// SIMATIC STEP 7 (V5.x) project Sald_Nozzle
// CPU: CPU 315-2 DP
// station: P_ADR_BUS
// station: Hardware
// station: SIMATIC 300(1)
// program: Programma S7(1)
// program: SINAMICS_S120_CU320

FUNCTION_BLOCK FB 16
AUTHOR : Cellini
VERSION : 0.1
BEGIN
// (block stored without names or comments; labels and parameter names are numbered)
NETWORK
TITLE =
      L     DIW [AR2,P#0.0];
      SLD   3;
      T     LD 28;
      L     P#DIX 2.0;
      T     LD 36;
      L     11;
M001: T     LW 34;
      L     PIW [LD 28];
      T     DIW [LD 36];
      L     LD 28;
      L     P#2.0;
      +D;
      T     LD 28;
      L     LD 36;
      L     P#2.0;
      +D;
      T     LD 36;
      L     LW 34;
      LOOP  M001;
NETWORK
TITLE =
      A     DIX [AR2,P#10.5];
      AN    DIX [AR2,P#10.4];
      =     DIX [AR2,P#45.1];
      A     DIX [AR2,P#11.0];
      A     DIX [AR2,P#11.1];
      A     DIX [AR2,P#11.2];
      AN    DIX [AR2,P#11.3];
      A     DIX [AR2,P#11.4];
      A     DIX [AR2,P#11.5];
      A     DIX [AR2,P#10.0];
      =     DIX [AR2,P#45.2];
      A     DIX [AR2,P#17.5];
      =     DIX [AR2,P#45.3];
      A     DIX [AR2,P#23.0];
      =     DIX [AR2,P#45.4];
      A     DIX [AR2,P#23.1];
      =     DIX [AR2,P#45.5];
      A     DIX [AR2,P#23.2];
      =     DIX [AR2,P#45.6];
      A     DIX [AR2,P#15.6];
      =     DIX [AR2,P#45.7];
      A     DIX [AR2,P#15.7];
      =     DIX [AR2,P#46.0];
      L     DID [AR2,P#18.0];
      T     DID [AR2,P#62.0];
NETWORK
TITLE =
      A     DIX [AR2,P#42.0];
      =     DIX [AR2,P#33.0];
      =     DIX [AR2,P#33.1];
      =     DIX [AR2,P#33.2];
      A     M 1.1;
      =     DIX [AR2,P#33.3];
      O     DIX [AR2,P#42.2];
      O     DIX [AR2,P#11.3];
      ON    DIX [AR2,P#10.0];
      R     DIX [AR2,P#42.3];
      R     DIX [AR2,P#44.0];
      R     DIX [AR2,P#44.1];
      R     DIX [AR2,P#42.4];
      R     DIX [AR2,P#44.2];
      R     DIX [AR2,P#44.3];
      R     DIX [AR2,P#42.5];
      R     DIX [AR2,P#42.6];
      R     DIX [AR2,P#32.3];
      R     DIX [AR2,P#33.6];
      AN    DIX [AR2,P#42.2];
      =     DIX [AR2,P#33.4];
      AN    DIX [AR2,P#42.7];
      =     DIX [AR2,P#33.5];
      A     DIX [AR2,P#42.1];
      =     DIX [AR2,P#33.7];
      A     DIX [AR2,P#10.1];
      =     DIX [AR2,P#32.2];
      L     DIW [AR2,P#60.0];
      T     DIW [AR2,P#40.0];
NETWORK
TITLE =
      A     DIX [AR2,P#42.3];
      A(;
      L     DID [AR2,P#48.0];
      L     50;
      <D;
      );
      A(;
      L     DID [AR2,P#48.0];
      L     -50;
      >D;
      );
      R     DIX [AR2,P#42.3];
      A     DIX [AR2,P#42.3];
      R     DIX [AR2,P#35.0];
      S     DIX [AR2,P#35.1];
      R     DIX [AR2,P#35.2];
      R     DIX [AR2,P#35.3];
      R     DIX [AR2,P#35.4];
      R     DIX [AR2,P#35.5];
      A     DIX [AR2,P#42.3];
      AN    DIX [AR2,P#44.0];
      AN    DIX [AR2,P#44.1];
      S     DIX [AR2,P#44.0];
      JCN   M002;
      L     DID [AR2,P#48.0];
      T     DID [AR2,P#28.0];
      L     W#16#8051;
      T     DIW [AR2,P#24.0];
      L     2;
      T     DIW [AR2,P#26.0];
M002: NOP   0;
      A     DIX [AR2,P#42.3];
      A     DIX [AR2,P#44.0];
      AN    DIX [AR2,P#44.1];
      A(;
      L     DID [AR2,P#28.0];
      L     DID [AR2,P#6.0];
      ==D;
      );
      A(;
      L     W#16#5051;
      L     DIW [AR2,P#2.0];
      ==I;
      );
      A(;
      L     DIW [AR2,P#26.0];
      L     DIW [AR2,P#4.0];
      ==I;
      );
      S     DIX [AR2,P#44.1];
      A     DIX [AR2,P#42.3];
      A     DIX [AR2,P#44.0];
      A     DIX [AR2,P#44.1];
      A(;
      L     DID [AR2,P#48.0];
      L     DID [AR2,P#6.0];
      ==D;
      );
      AN    DIX [AR2,P#33.6];
      S     DIX [AR2,P#33.6];
      JCN   M003;
      L     0;
      T     DIW [AR2,P#24.0];
      T     DIW [AR2,P#26.0];
      T     DID [AR2,P#28.0];
M003: NOP   0;
      A     DIX [AR2,P#10.2];
      FP    DIX [AR2,P#47.0];
      A     DIX [AR2,P#42.3];
      A     DIX [AR2,P#44.0];
      A     DIX [AR2,P#44.1];
      A     DIX [AR2,P#33.6];
      R     DIX [AR2,P#33.6];
      R     DIX [AR2,P#42.3];
      R     DIX [AR2,P#44.0];
      R     DIX [AR2,P#44.1];
NETWORK
TITLE =
      A     DIX [AR2,P#42.4];
      AN    DIX [AR2,P#44.2];
      AN    DIX [AR2,P#44.3];
      JCN   M005;
      L     DID [AR2,P#52.0];
      L     DID [AR2,P#18.0];
      -D;
      T     DID [AR2,P#56.0];
      L     0;
      <D;
      JCN   M004;
      L     DID [AR2,P#56.0];
      NEGD;
      T     DID [AR2,P#56.0];
M004: NOP   0;
      A(;
      L     DID [AR2,P#56.0];
      L     99;
      <=D;
      );
      R     DIX [AR2,P#42.4];
M005: NOP   0;
      A     DIX [AR2,P#42.4];
      R     DIX [AR2,P#35.0];
      R     DIX [AR2,P#35.1];
      R     DIX [AR2,P#35.2];
      R     DIX [AR2,P#35.3];
      R     DIX [AR2,P#35.4];
      R     DIX [AR2,P#35.5];
      A     DIX [AR2,P#42.4];
      AN    DIX [AR2,P#44.2];
      AN    DIX [AR2,P#44.3];
      S     DIX [AR2,P#44.2];
      JCN   M006;
      L     DID [AR2,P#52.0];
      T     DID [AR2,P#28.0];
      L     W#16#8051;
      T     DIW [AR2,P#24.0];
      L     0;
      T     DIW [AR2,P#26.0];
M006: NOP   0;
      A     DIX [AR2,P#42.4];
      A     DIX [AR2,P#44.2];
      AN    DIX [AR2,P#44.3];
      A(;
      L     DID [AR2,P#28.0];
      L     DID [AR2,P#6.0];
      ==D;
      );
      A(;
      L     W#16#5051;
      L     DIW [AR2,P#2.0];
      ==I;
      );
      A(;
      L     DIW [AR2,P#26.0];
      L     DIW [AR2,P#4.0];
      ==I;
      );
      S     DIX [AR2,P#44.3];
      A     DIX [AR2,P#42.4];
      A     DIX [AR2,P#44.2];
      A     DIX [AR2,P#44.3];
      A(;
      L     DID [AR2,P#52.0];
      L     DID [AR2,P#6.0];
      ==D;
      );
      AN    DIX [AR2,P#13.0];
      AN    DIX [AR2,P#13.1];
      AN    DIX [AR2,P#13.2];
      AN    DIX [AR2,P#13.3];
      AN    DIX [AR2,P#13.4];
      AN    DIX [AR2,P#13.5];
      AN    DIX [AR2,P#33.6];
      S     DIX [AR2,P#33.6];
      JCN   M007;
      L     0;
      T     DIW [AR2,P#24.0];
      T     DIW [AR2,P#26.0];
      T     DID [AR2,P#28.0];
M007: NOP   0;
      A     DIX [AR2,P#10.2];
      FP    DIX [AR2,P#47.1];
      A     DIX [AR2,P#42.4];
      A     DIX [AR2,P#44.2];
      A     DIX [AR2,P#44.3];
      A     DIX [AR2,P#33.6];
      R     DIX [AR2,P#33.6];
      R     DIX [AR2,P#42.4];
      R     DIX [AR2,P#44.2];
      R     DIX [AR2,P#44.3];
NETWORK
TITLE =
      A     DIX [AR2,P#42.5];
      FP    DIX [AR2,P#47.2];
      A     DIX [AR2,P#45.0];
      R     DIX [AR2,P#42.5];
      A     DIX [AR2,P#42.5];
      S     DIX [AR2,P#35.0];
      R     DIX [AR2,P#35.1];
      R     DIX [AR2,P#35.2];
      R     DIX [AR2,P#35.3];
      R     DIX [AR2,P#35.4];
      R     DIX [AR2,P#35.5];
      A     DIX [AR2,P#42.5];
      A     DIX [AR2,P#13.0];
      AN    DIX [AR2,P#13.1];
      AN    DIX [AR2,P#13.2];
      AN    DIX [AR2,P#13.3];
      AN    DIX [AR2,P#13.4];
      AN    DIX [AR2,P#13.5];
      AN    DIX [AR2,P#33.6];
      S     DIX [AR2,P#33.6];
      A     DIX [AR2,P#10.2];
      FP    DIX [AR2,P#47.3];
      A     DIX [AR2,P#42.5];
      A     DIX [AR2,P#33.6];
      R     DIX [AR2,P#33.6];
      R     DIX [AR2,P#42.5];
NETWORK
TITLE =
      A     DIX [AR2,P#43.0];
      A     DIX [AR2,P#10.3];
      AN    DIX [AR2,P#15.7];
      =     DIX [AR2,P#32.1];
      A     DIX [AR2,P#43.1];
      A     DIX [AR2,P#10.3];
      AN    DIX [AR2,P#15.6];
      =     DIX [AR2,P#32.0];
NETWORK
TITLE =
      A     DIX [AR2,P#42.6];
      FP    DIX [AR2,P#47.4];
      S     DIX [AR2,P#32.3];
      A     DIX [AR2,P#10.3];
      FP    DIX [AR2,P#47.5];
      R     DIX [AR2,P#32.3];
      R     DIX [AR2,P#42.6];
NETWORK
TITLE =
      L     DIW [AR2,P#0.0];
      SLD   3;
      T     LD 28;
      L     P#DIX 24.0;
      T     LD 36;
      L     9;
M008: T     LW 34;
      L     DIW [LD 36];
      T     PQW [LD 28];
      L     LD 28;
      L     P#2.0;
      +D;
      T     LD 28;
      L     LD 36;
      L     P#2.0;
      +D;
      T     LD 36;
      L     LW 34;
      LOOP  M008;
END_FUNCTION_BLOCK

FUNCTION_BLOCK FB 20
AUTHOR : Salvati
VERSION : 0.1
BEGIN
// (block stored without names or comments; labels and parameter names are numbered)
NETWORK
TITLE =
      TAR1  LD 0;
      TAR2  LD 4;
      LAR1  P#L 8.0;
      L     B#16#10;
      T     LB [AR1,P#0.0];
      L     B#16#2;
      T     LB [AR1,P#1.0];
      L     6;
      T     LW [AR1,P#2.0];
      L     0;
      T     LW [AR1,P#4.0];
      L     DIW 0;
      SLD   3;
      L     P#I 0.0;
      +D;
      T     LD [AR1,P#6.0];
      LAR1  P#L 18.0;
      L     B#16#10;
      T     LB [AR1,P#0.0];
      L     B#16#2;
      T     LB [AR1,P#1.0];
      L     6;
      T     LW [AR1,P#2.0];
      L     0;
      T     LW [AR1,P#4.0];
      L     P#DIX 2.0;
      T     LD [AR1,P#6.0];
      BLD   7;
      UC    SFC 20;
      {     P#L 8.0, P#L 34.0, P#L 18.0 };
      BLD   8;
      LAR1  LD 0;
      LAR2  LD 4;
NETWORK
TITLE =
      TAR1  LD 0;
      TAR2  LD 4;
      LAR1  P#L 8.0;
      L     B#16#10;
      T     LB [AR1,P#0.0];
      L     B#16#2;
      T     LB [AR1,P#1.0];
      L     6;
      T     LW [AR1,P#2.0];
      L     0;
      T     LW [AR1,P#4.0];
      L     DIW 0;
      SLD   3;
      L     P#Q 0.0;
      +D;
      T     LD [AR1,P#6.0];
      LAR1  P#L 18.0;
      L     B#16#10;
      T     LB [AR1,P#0.0];
      L     B#16#2;
      T     LB [AR1,P#1.0];
      L     6;
      T     LW [AR1,P#2.0];
      L     0;
      T     LW [AR1,P#4.0];
      L     P#DIX 8.0;
      T     LD [AR1,P#6.0];
      BLD   7;
      UC    SFC 20;
      {     P#L 8.0, P#L 34.0, P#L 18.0 };
      BLD   8;
      LAR1  LD 0;
      LAR2  LD 4;
NETWORK
TITLE =
      A     DIX 14.3;
      A     M 1.5;
      JCN   M001;
      L     DIB 18;
      L     1;
      +I;
      T     DIB 18;
M001: NOP   0;
      A     DIX 14.0;
      AN    DIX 15.0;
      AN    DIX 14.3;
      S     DIX 14.3;
      R     DIX 8.4;
      JCN   M002;
      L     0;
      T     DIB 18;
M002: NOP   0;
      A     DIX 14.0;
      A     DIX 14.3;
      AN    DIX 2.4;
      AN    DIX 14.4;
      S     DIX 14.4;
      A     DIX 14.0;
      A     DIX 14.4;
      A     DIX 2.7;
      A     DIX 2.0;
      AN    DIX 14.5;
      S     DIX 14.5;
      R     DIX 14.1;
      R     DIX 14.2;
      S     DIX 8.0;
      R     DIX 8.7;
      JC    M003;
      JU    M004;
M003: NOP   0;
      L     0;
      T     DIB 10;
      T     DIB 11;
      T     DIB 13;
      L     1;
      T     DIB 12;
      L     1;
      T     DIB 9;
M004: NOP   0;
      A     DIX 14.0;
      A     DIX 14.5;
      A     DIX 2.1;
      A     DIX 2.3;
      O;
      A(;
      L     DIB 18;
      L     10;
      >=I;
      );
      R     DIX 14.3;
      R     DIX 14.4;
      R     DIX 14.5;
      R     DIX 8.0;
      R     DIX 14.0;
      S     DIX 14.2;
      JCN   M005;
      L     0;
      T     DIB 18;
M005: NOP   0;
      A     DIX 14.0;
      A     DIX 14.5;
      A     DIX 2.1;
      A     DIX 2.2;
      R     DIX 14.3;
      R     DIX 14.4;
      R     DIX 14.5;
      R     DIX 8.0;
      R     DIX 14.0;
      S     DIX 14.1;
      JC    M006;
      JU    M007;
M006: L     DIB 3;
      T     DIB 16;
M007: NOP   0;
NETWORK
TITLE =
      A     DIX 15.3;
      A     M 1.5;
      JCN   M008;
      L     DIB 18;
      L     1;
      +I;
      T     DIB 18;
M008: NOP   0;
      A     DIX 15.0;
      AN    DIX 14.0;
      AN    DIX 15.3;
      S     DIX 15.3;
      R     DIX 8.4;
      JCN   M009;
      L     0;
      T     DIB 18;
M009: NOP   0;
      A     DIX 15.0;
      A     DIX 15.3;
      AN    DIX 2.4;
      AN    DIX 15.4;
      S     DIX 15.4;
      A     DIX 15.0;
      A     DIX 15.4;
      A     DIX 2.7;
      A     DIX 2.0;
      AN    DIX 15.5;
      S     DIX 15.5;
      R     DIX 15.1;
      R     DIX 15.2;
      S     DIX 8.0;
      R     DIX 8.7;
      JC    M010;
      JU    M011;
M010: NOP   0;
      L     0;
      T     DIB 10;
      T     DIB 11;
      T     DIB 13;
      L     1;
      T     DIB 12;
      L     2;
      T     DIB 9;
M011: NOP   0;
      A     DIX 15.0;
      A     DIX 15.5;
      A     DIX 2.1;
      A     DIX 2.5;
      AN    DIX 15.6;
      S     DIX 15.6;
      S     DIX 8.6;
      JC    M012;
      JU    M013;
M012: NOP   0;
      L     DIB 17;
      T     DIB 9;
M013: NOP   0;
      A     DIX 15.0;
      A     DIX 15.6;
      A     DIX 2.1;
      A     DIX 2.3;
      O;
      A(;
      L     DIB 18;
      L     10;
      >=I;
      );
      R     DIX 15.3;
      R     DIX 15.4;
      R     DIX 15.5;
      R     DIX 15.6;
      R     DIX 8.0;
      R     DIX 8.6;
      R     DIX 15.0;
      S     DIX 15.2;
      JCN   M014;
      L     0;
      T     DIB 18;
M014: NOP   0;
      A     DIX 15.0;
      A     DIX 15.6;
      A     DIX 2.1;
      A     DIX 2.2;
      R     DIX 15.3;
      R     DIX 15.4;
      R     DIX 15.5;
      R     DIX 15.6;
      R     DIX 8.0;
      R     DIX 8.6;
      R     DIX 15.0;
      S     DIX 15.1;
NETWORK
TITLE =
      A     DIX 20.3;
      A     M 1.5;
      JCN   M015;
      L     DIB 24;
      L     1;
      +I;
      T     DIB 24;
M015: NOP   0;
      A     DIX 20.0;
      AN    DIX 21.0;
      AN    DIX 14.0;
      AN    DIX 15.0;
      AN    DIX 20.3;
      S     DIX 20.3;
      S     DIX 8.4;
      JCN   M016;
      L     0;
      T     DIB 24;
M016: NOP   0;
      A     DIX 20.0;
      A     DIX 20.3;
      A     DIX 2.4;
      AN    DIX 20.4;
      S     DIX 20.4;
      A     DIX 20.0;
      A     DIX 20.4;
      A     DIX 2.7;
      A     DIX 2.0;
      AN    DIX 20.5;
      S     DIX 20.5;
      R     DIX 20.1;
      R     DIX 20.2;
      S     DIX 8.0;
      R     DIX 8.7;
      JC    M017;
      JU    M018;
M017: NOP   0;
      L     0;
      T     DIB 10;
      T     DIB 11;
      T     DIB 13;
      L     1;
      T     DIB 12;
      L     1;
      T     DIB 9;
M018: NOP   0;
      A     DIX 20.0;
      A     DIX 20.5;
      A     DIX 2.1;
      A     DIX 2.3;
      O;
      A(;
      L     DIB 24;
      L     10;
      >=I;
      );
      R     DIX 20.3;
      R     DIX 20.4;
      R     DIX 20.5;
      R     DIX 8.0;
      R     DIX 20.0;
      S     DIX 20.2;
      JCN   M019;
      L     0;
      T     DIB 24;
M019: NOP   0;
      A     DIX 20.0;
      A     DIX 20.5;
      A     DIX 2.1;
      A     DIX 2.2;
      R     DIX 20.3;
      R     DIX 20.4;
      R     DIX 20.5;
      R     DIX 8.0;
      R     DIX 20.0;
      S     DIX 20.1;
      JC    M020;
      JU    M021;
M020: L     DIB 3;
      T     DIB 22;
M021: NOP   0;
NETWORK
TITLE =
      A     DIX 21.3;
      A     M 1.5;
      JCN   M022;
      L     DIB 24;
      L     1;
      +I;
      T     DIB 24;
M022: NOP   0;
      A     DIX 21.0;
      AN    DIX 20.0;
      AN    DIX 14.0;
      AN    DIX 15.0;
      AN    DIX 21.3;
      S     DIX 21.3;
      S     DIX 8.4;
      JCN   M023;
      L     0;
      T     DIB 24;
M023: NOP   0;
      A     DIX 21.0;
      A     DIX 21.3;
      A     DIX 2.4;
      AN    DIX 21.4;
      S     DIX 21.4;
      A     DIX 21.0;
      A     DIX 21.4;
      A     DIX 2.7;
      A     DIX 2.0;
      AN    DIX 21.5;
      S     DIX 21.5;
      R     DIX 21.1;
      R     DIX 21.2;
      S     DIX 8.0;
      R     DIX 8.7;
      JC    M024;
      JU    M025;
M024: NOP   0;
      L     0;
      T     DIB 10;
      T     DIB 11;
      T     DIB 13;
      L     1;
      T     DIB 12;
      L     2;
      T     DIB 9;
M025: NOP   0;
      A     DIX 21.0;
      A     DIX 21.5;
      A     DIX 2.1;
      A     DIX 2.5;
      AN    DIX 21.6;
      S     DIX 21.6;
      S     DIX 8.6;
      JC    M026;
      JU    M027;
M026: NOP   0;
      L     DIB 23;
      T     DIB 9;
M027: NOP   0;
      A     DIX 21.0;
      A     DIX 21.6;
      A     DIX 2.1;
      A     DIX 2.3;
      O;
      A(;
      L     DIB 24;
      L     10;
      >=I;
      );
      R     DIX 21.3;
      R     DIX 21.4;
      R     DIX 21.5;
      R     DIX 21.6;
      R     DIX 8.0;
      R     DIX 8.6;
      R     DIX 21.0;
      S     DIX 21.2;
      JCN   M028;
      L     0;
      T     DIB 24;
M028: NOP   0;
      A     DIX 21.0;
      A     DIX 21.6;
      A     DIX 2.1;
      A     DIX 2.2;
      R     DIX 21.3;
      R     DIX 21.4;
      R     DIX 21.5;
      R     DIX 21.6;
      R     DIX 8.0;
      R     DIX 8.6;
      R     DIX 21.0;
      S     DIX 21.1;
NETWORK
TITLE =
      TAR1  LD 0;
      TAR2  LD 4;
      LAR1  P#L 8.0;
      L     B#16#10;
      T     LB [AR1,P#0.0];
      L     B#16#2;
      T     LB [AR1,P#1.0];
      L     6;
      T     LW [AR1,P#2.0];
      L     0;
      T     LW [AR1,P#4.0];
      L     P#DIX 8.0;
      T     LD [AR1,P#6.0];
      LAR1  P#L 18.0;
      L     B#16#10;
      T     LB [AR1,P#0.0];
      L     B#16#2;
      T     LB [AR1,P#1.0];
      L     6;
      T     LW [AR1,P#2.0];
      L     0;
      T     LW [AR1,P#4.0];
      L     DIW 0;
      SLD   3;
      L     P#Q 0.0;
      +D;
      T     LD [AR1,P#6.0];
      BLD   7;
      UC    SFC 20;
      {     P#L 8.0, P#L 34.0, P#L 18.0 };
      BLD   8;
      LAR1  LD 0;
      LAR2  LD 4;
END_FUNCTION_BLOCK

FUNCTION_BLOCK FB 24
VERSION : 0.1
BEGIN
// (block stored without names or comments; labels and parameter names are numbered)
NETWORK
TITLE =
      L     DID [AR2,P#0.0];
      L     8;
      +I;
      SLD   3;
      T     MD 100;
      L     PIW [MD 100];
      T     DIW 52;
      L     MD 100;
      SRW   3;
      L     2;
      +D;
      SLW   3;
      T     MD 100;
      L     PIW [MD 100];
      T     DIW [AR2,P#46.0];
      L     MD 100;
      SRW   3;
      L     2;
      +D;
      SLW   3;
      T     MD 100;
      L     PIW [MD 100];
      T     DIW 64;
      L     MD 100;
      SRW   3;
      L     2;
      +D;
      SLW   3;
      T     MD 100;
      L     PIW [MD 100];
      T     DIW 62;
      L     MD 100;
      SRW   3;
      L     2;
      +D;
      SLW   3;
      T     MD 100;
      L     PID [MD 100];
      T     DID [AR2,P#36.0];
      L     MD 100;
      SRW   3;
      L     4;
      +D;
      SLW   3;
      T     MD 100;
      L     PIW [MD 100];
      T     DIW 54;
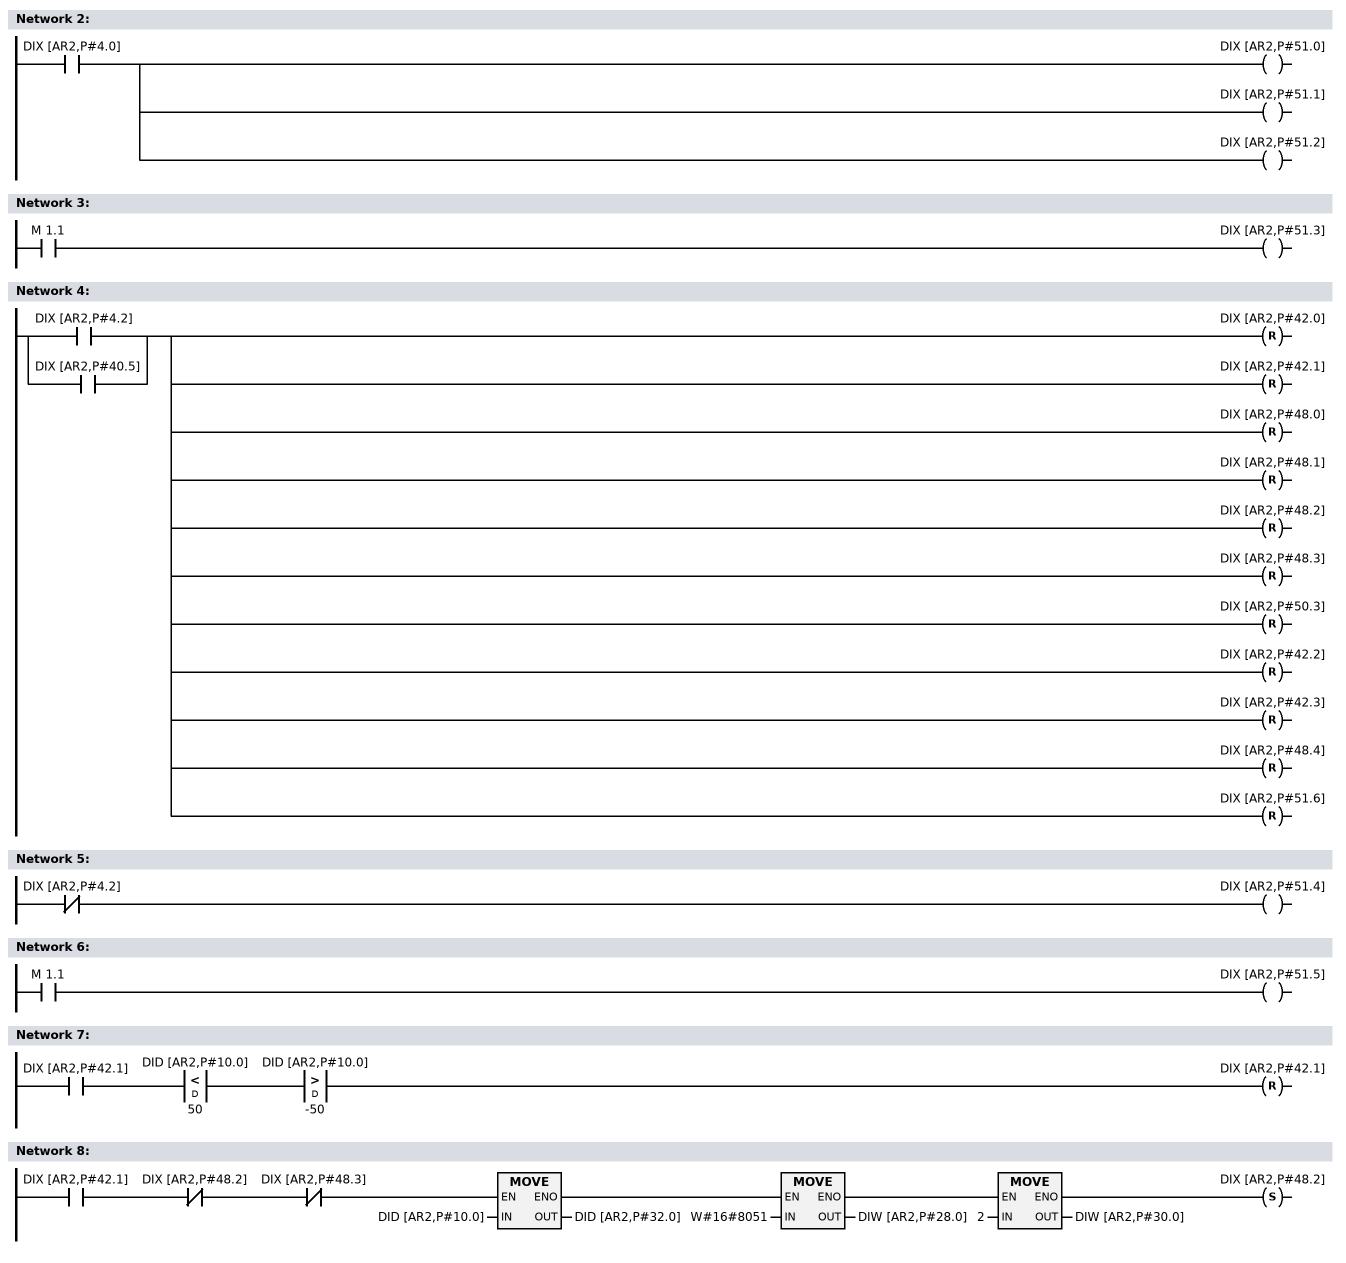
NETWORK
TITLE =
      A     DIX [AR2,P#4.0];
      =     DIX [AR2,P#51.0];
      =     DIX [AR2,P#51.1];
      =     DIX [AR2,P#51.2];
NETWORK
TITLE =
      A     M 1.1;
      =     DIX [AR2,P#51.3];
NETWORK
TITLE =
      O     DIX [AR2,P#4.2];
      O     DIX [AR2,P#40.5];
      R     DIX [AR2,P#42.0];
      R     DIX [AR2,P#42.1];
      R     DIX [AR2,P#48.0];
      R     DIX [AR2,P#48.1];
      R     DIX [AR2,P#48.2];
      R     DIX [AR2,P#48.3];
      R     DIX [AR2,P#50.3];
      R     DIX [AR2,P#42.2];
      R     DIX [AR2,P#42.3];
      R     DIX [AR2,P#48.4];
      R     DIX [AR2,P#51.6];
NETWORK
TITLE =
      AN    DIX [AR2,P#4.2];
      =     DIX [AR2,P#51.4];
NETWORK
TITLE =
      A     M 1.1;
      =     DIX [AR2,P#51.5];
NETWORK
TITLE =
      A     DIX [AR2,P#42.1];
      A(;
      L     DID [AR2,P#10.0];
      L     50;
      <D;
      );
      A(;
      L     DID [AR2,P#10.0];
      L     -50;
      >D;
      );
      R     DIX [AR2,P#42.1];
NETWORK
TITLE =
      A(;
      A(;
      A     DIX [AR2,P#42.1];
      AN    DIX [AR2,P#48.2];
      AN    DIX [AR2,P#48.3];
      JNB   M001;
      L     DID [AR2,P#10.0];
      T     DID [AR2,P#32.0];
      SET;
      SAVE;
      CLR;
M001: A     BR;
      );
      JNB   M002;
      L     W#16#8051;
      T     DIW [AR2,P#28.0];
      SET;
      SAVE;
      CLR;
M002: A     BR;
      );
      JNB   M003;
      L     2;
      T     DIW [AR2,P#30.0];
      SET;
      SAVE;
      CLR;
M003: A     BR;
      S     DIX [AR2,P#48.2];
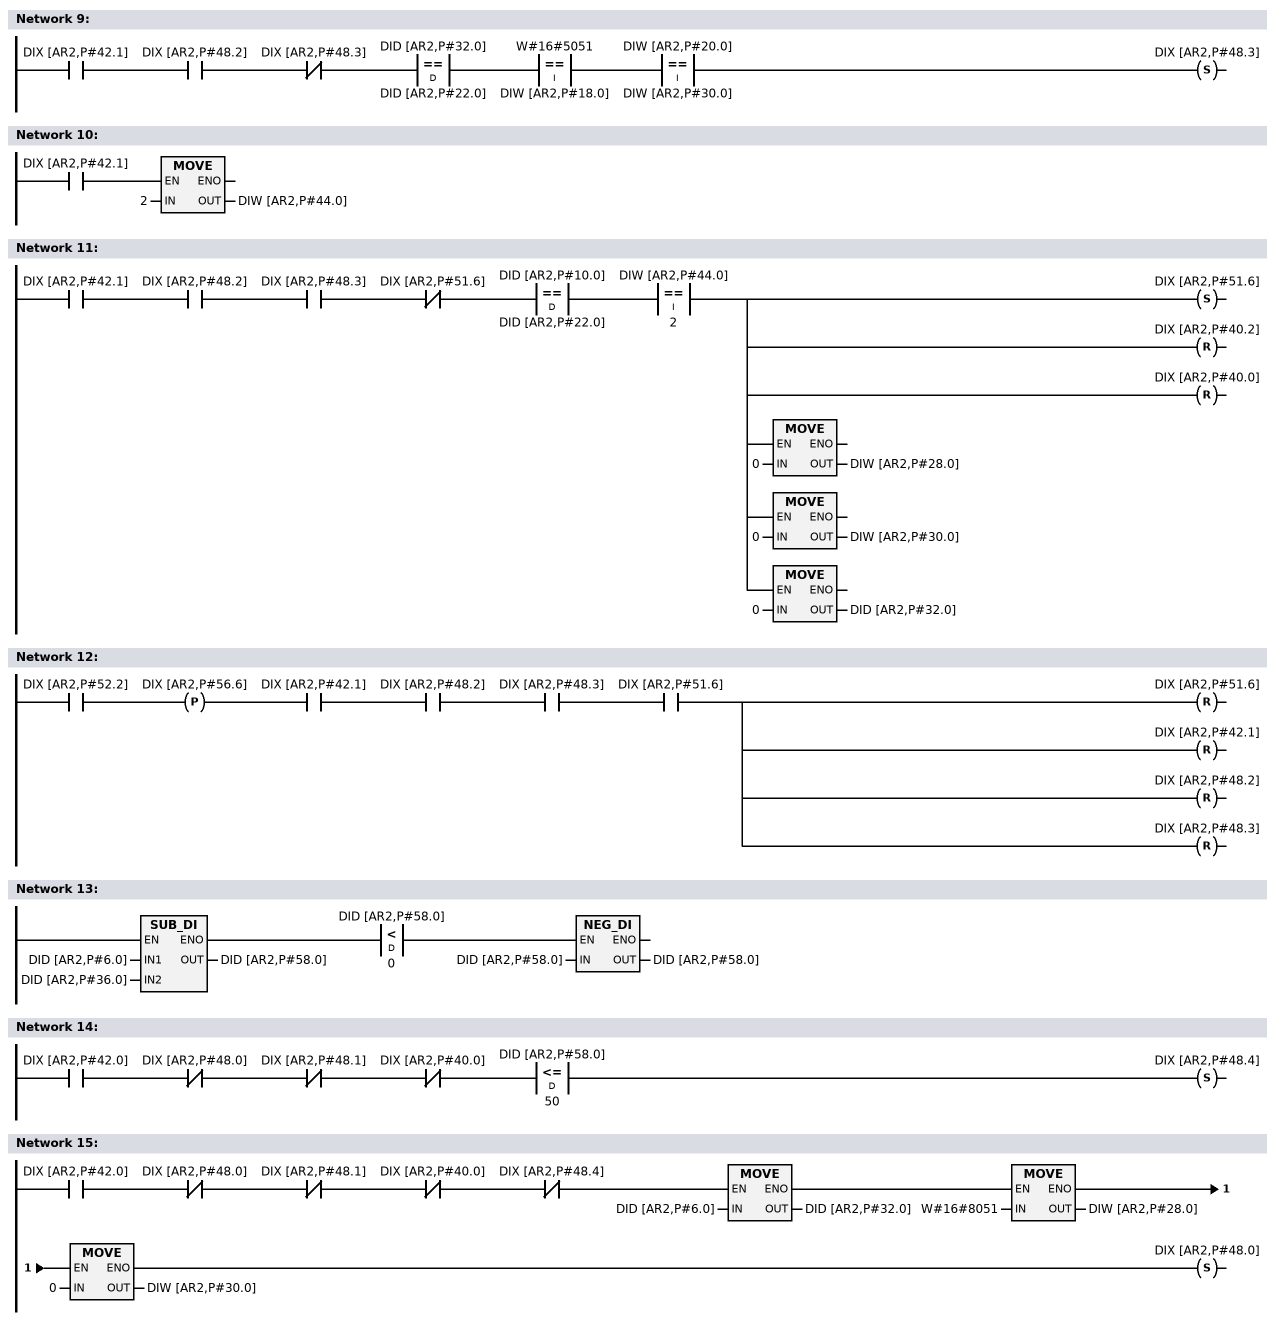
NETWORK
TITLE =
      A     DIX [AR2,P#42.1];
      A     DIX [AR2,P#48.2];
      AN    DIX [AR2,P#48.3];
      A(;
      L     DID [AR2,P#32.0];
      L     DID [AR2,P#22.0];
      ==D;
      );
      A(;
      L     W#16#5051;
      L     DIW [AR2,P#18.0];
      ==I;
      );
      A(;
      L     DIW [AR2,P#20.0];
      L     DIW [AR2,P#30.0];
      ==I;
      );
      S     DIX [AR2,P#48.3];
NETWORK
TITLE =
      A     DIX [AR2,P#42.1];
      JNB   M004;
      L     2;
      T     DIW [AR2,P#44.0];
M004: NOP   0;
NETWORK
TITLE =
      A     DIX [AR2,P#42.1];
      A     DIX [AR2,P#48.2];
      A     DIX [AR2,P#48.3];
      AN    DIX [AR2,P#51.6];
      A(;
      L     DID [AR2,P#10.0];
      L     DID [AR2,P#22.0];
      ==D;
      );
      A(;
      L     DIW [AR2,P#44.0];
      L     2;
      ==I;
      );
      =     L 0.0;
      A     L 0.0;
      BLD   102;
      S     DIX [AR2,P#51.6];
      A     L 0.0;
      BLD   102;
      R     DIX [AR2,P#40.2];
      A     L 0.0;
      BLD   102;
      R     DIX [AR2,P#40.0];
      A     L 0.0;
      JNB   M005;
      L     0;
      T     DIW [AR2,P#28.0];
M005: NOP   0;
      A     L 0.0;
      JNB   M006;
      L     0;
      T     DIW [AR2,P#30.0];
M006: NOP   0;
      A     L 0.0;
      JNB   M007;
      L     0;
      T     DID [AR2,P#32.0];
M007: NOP   0;
NETWORK
TITLE =
      A     DIX [AR2,P#52.2];
      FP    DIX [AR2,P#56.6];
      A     DIX [AR2,P#42.1];
      A     DIX [AR2,P#48.2];
      A     DIX [AR2,P#48.3];
      A     DIX [AR2,P#51.6];
      R     DIX [AR2,P#51.6];
      R     DIX [AR2,P#42.1];
      R     DIX [AR2,P#48.2];
      R     DIX [AR2,P#48.3];
NETWORK
TITLE =
      A(;
      L     DID [AR2,P#6.0];
      L     DID [AR2,P#36.0];
      -D;
      T     DID [AR2,P#58.0];
      AN    OV;
      SAVE;
      CLR;
      A     BR;
      );
      A(;
      L     DID [AR2,P#58.0];
      L     0;
      <D;
      );
      JNB   M008;
      L     DID [AR2,P#58.0];
      NEGD;
      T     DID [AR2,P#58.0];
M008: NOP   0;
NETWORK
TITLE =
      A     DIX [AR2,P#42.0];
      AN    DIX [AR2,P#48.0];
      AN    DIX [AR2,P#48.1];
      AN    DIX [AR2,P#40.0];
      A(;
      L     DID [AR2,P#58.0];
      L     50;
      <=D;
      );
      S     DIX [AR2,P#48.4];
NETWORK
TITLE =
      A(;
      A(;
      A     DIX [AR2,P#42.0];
      AN    DIX [AR2,P#48.0];
      AN    DIX [AR2,P#48.1];
      AN    DIX [AR2,P#40.0];
      AN    DIX [AR2,P#48.4];
      JNB   M009;
      L     DID [AR2,P#6.0];
      T     DID [AR2,P#32.0];
      SET;
      SAVE;
      CLR;
M009: A     BR;
      );
      JNB   M010;
      L     W#16#8051;
      T     DIW [AR2,P#28.0];
      SET;
      SAVE;
      CLR;
M010: A     BR;
      );
      JNB   M011;
      L     0;
      T     DIW [AR2,P#30.0];
      SET;
      SAVE;
      CLR;
M011: A     BR;
      S     DIX [AR2,P#48.0];
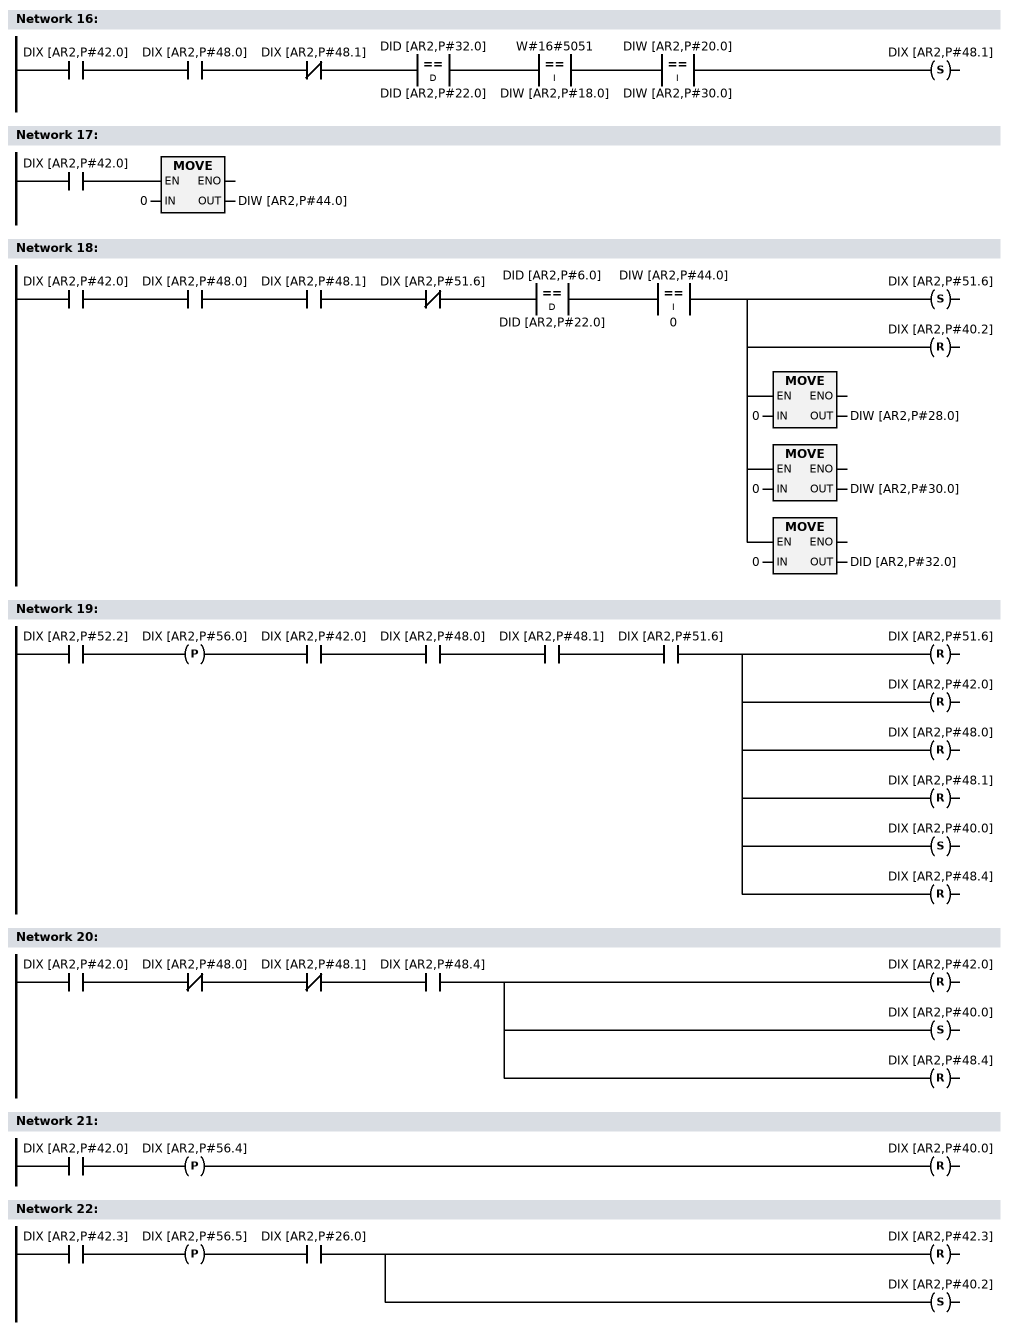
NETWORK
TITLE =
      A     DIX [AR2,P#42.0];
      A     DIX [AR2,P#48.0];
      AN    DIX [AR2,P#48.1];
      A(;
      L     DID [AR2,P#32.0];
      L     DID [AR2,P#22.0];
      ==D;
      );
      A(;
      L     W#16#5051;
      L     DIW [AR2,P#18.0];
      ==I;
      );
      A(;
      L     DIW [AR2,P#20.0];
      L     DIW [AR2,P#30.0];
      ==I;
      );
      S     DIX [AR2,P#48.1];
NETWORK
TITLE =
      A     DIX [AR2,P#42.0];
      JNB   M012;
      L     0;
      T     DIW [AR2,P#44.0];
M012: NOP   0;
NETWORK
TITLE =
      A     DIX [AR2,P#42.0];
      A     DIX [AR2,P#48.0];
      A     DIX [AR2,P#48.1];
      AN    DIX [AR2,P#51.6];
      A(;
      L     DID [AR2,P#6.0];
      L     DID [AR2,P#22.0];
      ==D;
      );
      A(;
      L     DIW [AR2,P#44.0];
      L     0;
      ==I;
      );
      =     L 0.0;
      A     L 0.0;
      BLD   102;
      S     DIX [AR2,P#51.6];
      A     L 0.0;
      BLD   102;
      R     DIX [AR2,P#40.2];
      A     L 0.0;
      JNB   M013;
      L     0;
      T     DIW [AR2,P#28.0];
M013: NOP   0;
      A     L 0.0;
      JNB   M014;
      L     0;
      T     DIW [AR2,P#30.0];
M014: NOP   0;
      A     L 0.0;
      JNB   M015;
      L     0;
      T     DID [AR2,P#32.0];
M015: NOP   0;
NETWORK
TITLE =
      A     DIX [AR2,P#52.2];
      FP    DIX [AR2,P#56.0];
      A     DIX [AR2,P#42.0];
      A     DIX [AR2,P#48.0];
      A     DIX [AR2,P#48.1];
      A     DIX [AR2,P#51.6];
      R     DIX [AR2,P#51.6];
      R     DIX [AR2,P#42.0];
      R     DIX [AR2,P#48.0];
      R     DIX [AR2,P#48.1];
      S     DIX [AR2,P#40.0];
      R     DIX [AR2,P#48.4];
NETWORK
TITLE =
      A     DIX [AR2,P#42.0];
      AN    DIX [AR2,P#48.0];
      AN    DIX [AR2,P#48.1];
      A     DIX [AR2,P#48.4];
      R     DIX [AR2,P#42.0];
      S     DIX [AR2,P#40.0];
      R     DIX [AR2,P#48.4];
NETWORK
TITLE =
      A     DIX [AR2,P#42.0];
      FP    DIX [AR2,P#56.4];
      R     DIX [AR2,P#40.0];
NETWORK
TITLE =
      A     DIX [AR2,P#42.3];
      FP    DIX [AR2,P#56.5];
      A     DIX [AR2,P#26.0];
      R     DIX [AR2,P#42.3];
      S     DIX [AR2,P#40.2];
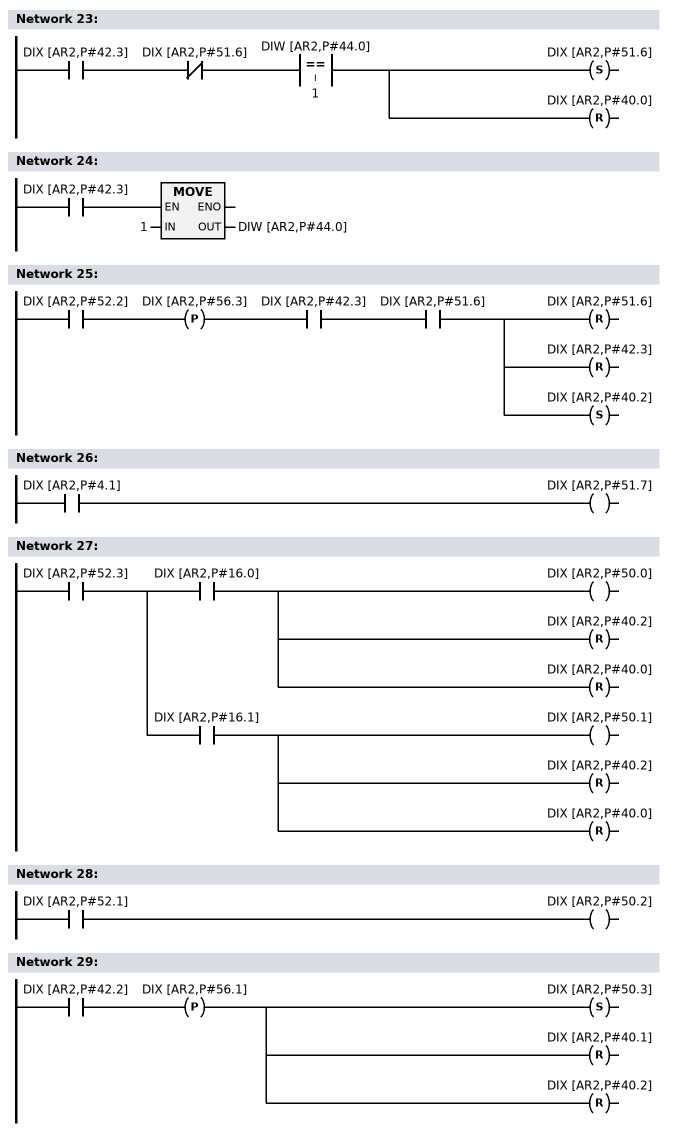
NETWORK
TITLE =
      A     DIX [AR2,P#42.3];
      AN    DIX [AR2,P#51.6];
      A(;
      L     DIW [AR2,P#44.0];
      L     1;
      ==I;
      );
      S     DIX [AR2,P#51.6];
      R     DIX [AR2,P#40.0];
NETWORK
TITLE =
      A     DIX [AR2,P#42.3];
      JNB   M016;
      L     1;
      T     DIW [AR2,P#44.0];
M016: NOP   0;
NETWORK
TITLE =
      A     DIX [AR2,P#52.2];
      FP    DIX [AR2,P#56.3];
      A     DIX [AR2,P#42.3];
      A     DIX [AR2,P#51.6];
      R     DIX [AR2,P#51.6];
      R     DIX [AR2,P#42.3];
      S     DIX [AR2,P#40.2];
NETWORK
TITLE =
      A     DIX [AR2,P#4.1];
      =     DIX [AR2,P#51.7];
NETWORK
TITLE =
      A     DIX [AR2,P#52.3];
      =     L 0.0;
      A     L 0.0;
      A     DIX [AR2,P#16.0];
      =     DIX [AR2,P#50.0];
      R     DIX [AR2,P#40.2];
      R     DIX [AR2,P#40.0];
      A     L 0.0;
      A     DIX [AR2,P#16.1];
      =     DIX [AR2,P#50.1];
      R     DIX [AR2,P#40.2];
      R     DIX [AR2,P#40.0];
NETWORK
TITLE =
      A     DIX [AR2,P#52.1];
      =     DIX [AR2,P#50.2];
NETWORK
TITLE =
      A     DIX [AR2,P#42.2];
      FP    DIX [AR2,P#56.1];
      S     DIX [AR2,P#50.3];
      R     DIX [AR2,P#40.1];
      R     DIX [AR2,P#40.2];
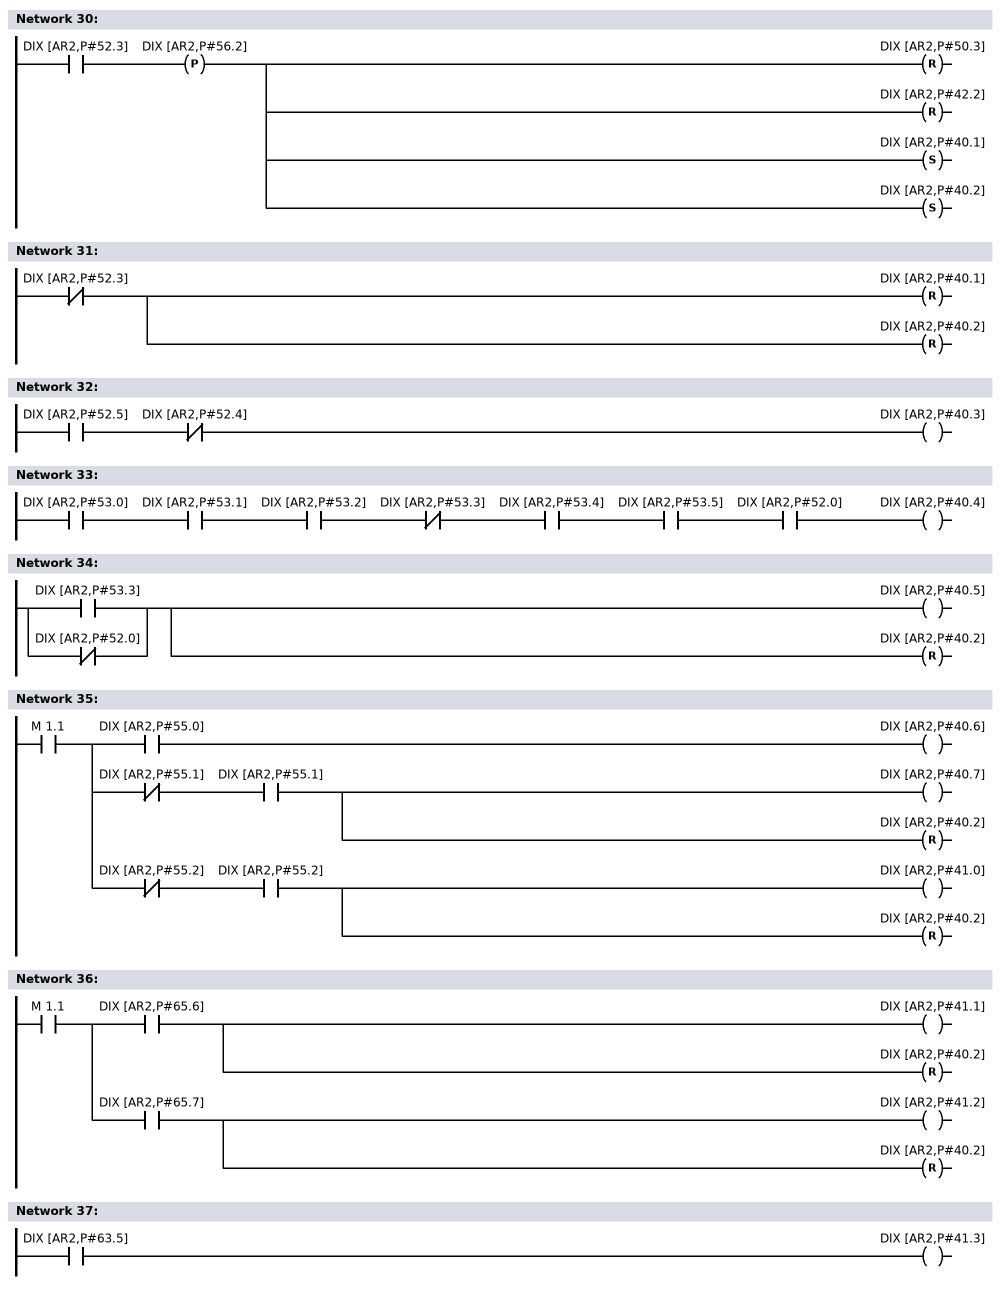
NETWORK
TITLE =
      A     DIX [AR2,P#52.3];
      FP    DIX [AR2,P#56.2];
      R     DIX [AR2,P#50.3];
      R     DIX [AR2,P#42.2];
      S     DIX [AR2,P#40.1];
      S     DIX [AR2,P#40.2];
NETWORK
TITLE =
      AN    DIX [AR2,P#52.3];
      R     DIX [AR2,P#40.1];
      R     DIX [AR2,P#40.2];
NETWORK
TITLE =
      A     DIX [AR2,P#52.5];
      AN    DIX [AR2,P#52.4];
      =     DIX [AR2,P#40.3];
NETWORK
TITLE =
      A     DIX [AR2,P#53.0];
      A     DIX [AR2,P#53.1];
      A     DIX [AR2,P#53.2];
      AN    DIX [AR2,P#53.3];
      A     DIX [AR2,P#53.4];
      A     DIX [AR2,P#53.5];
      A     DIX [AR2,P#52.0];
      =     DIX [AR2,P#40.4];
NETWORK
TITLE =
      O     DIX [AR2,P#53.3];
      ON    DIX [AR2,P#52.0];
      =     DIX [AR2,P#40.5];
      R     DIX [AR2,P#40.2];
NETWORK
TITLE =
      A     M 1.1;
      =     L 0.0;
      A     L 0.0;
      A     DIX [AR2,P#55.0];
      =     DIX [AR2,P#40.6];
      A     L 0.0;
      AN    DIX [AR2,P#55.1];
      A     DIX [AR2,P#55.1];
      =     DIX [AR2,P#40.7];
      R     DIX [AR2,P#40.2];
      A     L 0.0;
      AN    DIX [AR2,P#55.2];
      A     DIX [AR2,P#55.2];
      =     DIX [AR2,P#41.0];
      R     DIX [AR2,P#40.2];
NETWORK
TITLE =
      A     M 1.1;
      =     L 0.0;
      A     L 0.0;
      A     DIX [AR2,P#65.6];
      =     DIX [AR2,P#41.1];
      R     DIX [AR2,P#40.2];
      A     L 0.0;
      A     DIX [AR2,P#65.7];
      =     DIX [AR2,P#41.2];
      R     DIX [AR2,P#40.2];
NETWORK
TITLE =
      A     DIX [AR2,P#63.5];
      =     DIX [AR2,P#41.3];
NETWORK
TITLE =
      L     DID [AR2,P#0.0];
      L     8;
      +I;
      SLD   3;
      T     MD 100;
      L     DIW 50;
      T     PQW [MD 100];
      L     MD 100;
      SRW   3;
      L     2;
      +D;
      SLW   3;
      T     MD 100;
      L     DIW [AR2,P#44.0];
      T     PQW [MD 100];
      L     MD 100;
      SRW   3;
      L     6;
      +D;
      SLW   3;
      T     MD 100;
      L     DIW [AR2,P#14.0];
      T     PQW [MD 100];
END_FUNCTION_BLOCK

// FC 7: know-how protected block, not included

FUNCTION FC 11 : VOID
VERSION : 0.1
BEGIN
// (block stored without names or comments; labels and parameter names are numbered)
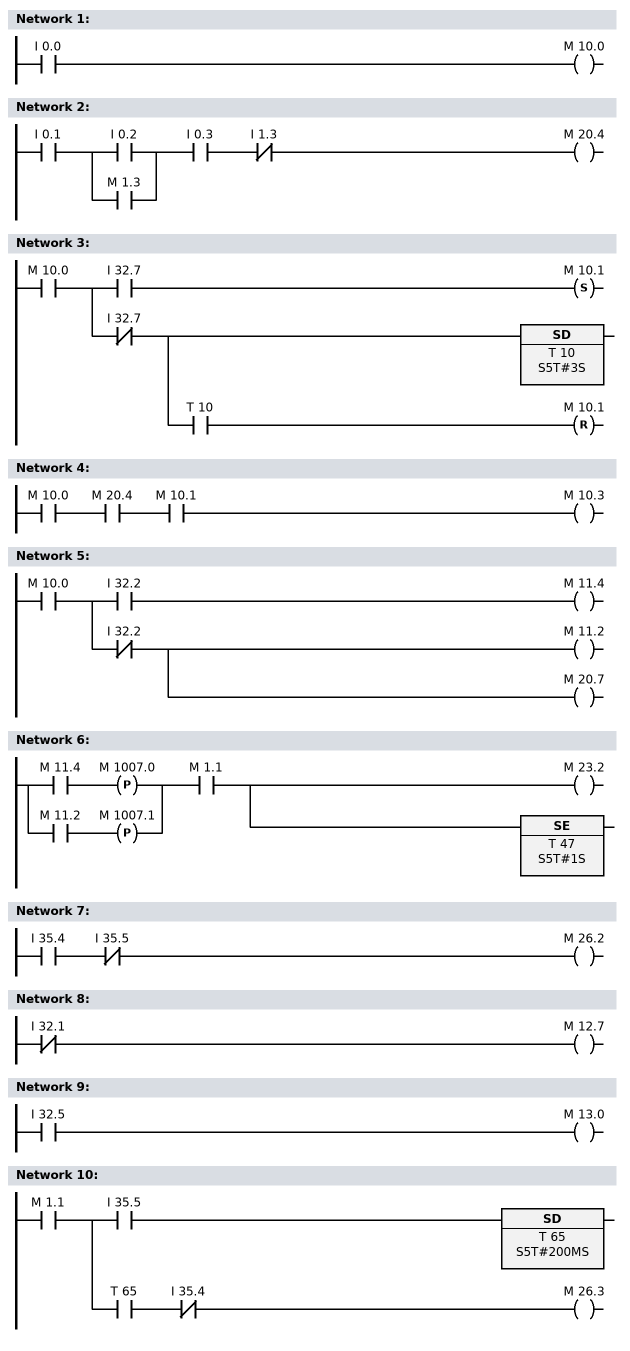
NETWORK
TITLE =
      A     I 0.0;
      =     M 10.0;
NETWORK
TITLE =
      A     I 0.1;
      A(;
      O     I 0.2;
      O     M 1.3;
      );
      A     I 0.3;
      AN    I 1.3;
      =     M 20.4;
NETWORK
TITLE =
      A     M 10.0;
      =     L 2.0;
      A     L 2.0;
      A     I 32.7;
      S     M 10.1;
      A     L 2.0;
      AN    I 32.7;
      =     L 2.1;
      A     L 2.1;
      BLD   102;
      L     S5T#3S;
      SD    T 10;
      A     L 2.1;
      A     T 10;
      R     M 10.1;
NETWORK
TITLE =
      A     M 10.0;
      A     M 20.4;
      A     M 10.1;
      =     M 10.3;
NETWORK
TITLE =
      A     M 10.0;
      =     L 2.0;
      A     L 2.0;
      A     I 32.2;
      =     M 11.4;
      A     L 2.0;
      AN    I 32.2;
      =     M 11.2;
      =     M 20.7;
NETWORK
TITLE =
      A(;
      A     M 11.4;
      FP    M 1007.0;
      O(;
      A     M 11.2;
      FP    M 1007.1;
      );
      );
      A     M 1.1;
      =     M 23.2;
      L     S5T#1S;
      SE    T 47;
NETWORK
TITLE =
      A     I 35.4;
      AN    I 35.5;
      =     M 26.2;
NETWORK
TITLE =
      AN    I 32.1;
      =     M 12.7;
NETWORK
TITLE =
      A     I 32.5;
      =     M 13.0;
NETWORK
TITLE =
      A     M 1.1;
      =     L 2.0;
      A     L 2.0;
      A     I 35.5;
      L     S5T#200MS;
      SD    T 65;
      A     L 2.0;
      A     T 65;
      AN    I 35.4;
      =     M 26.3;
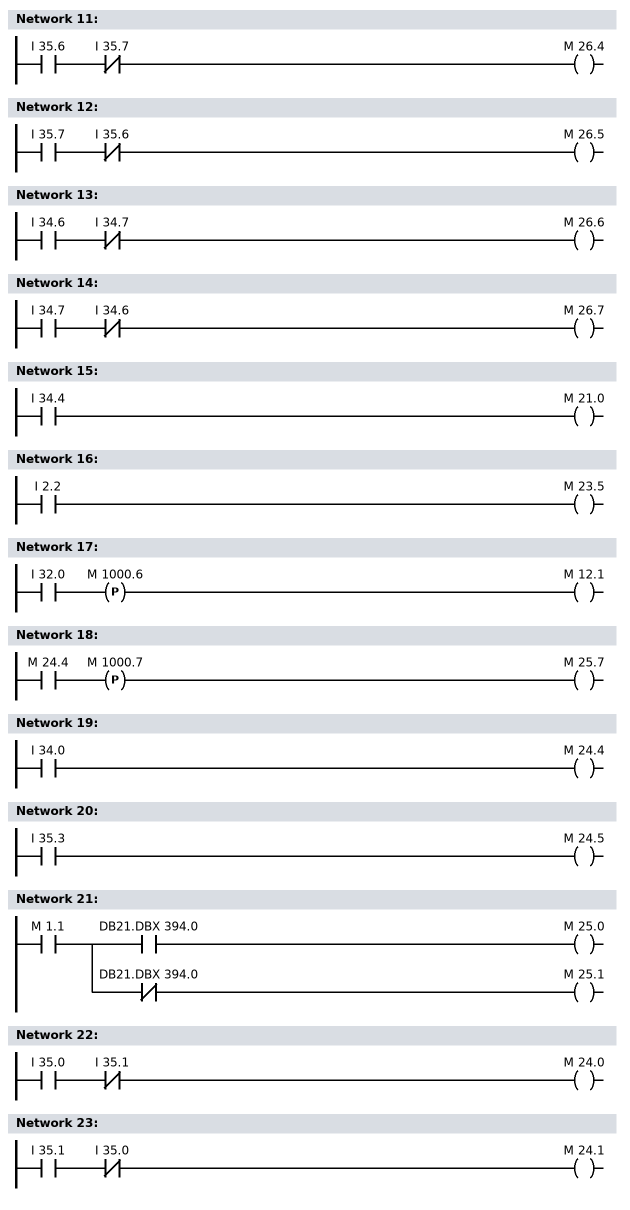
NETWORK
TITLE =
      A     I 35.6;
      AN    I 35.7;
      =     M 26.4;
NETWORK
TITLE =
      A     I 35.7;
      AN    I 35.6;
      =     M 26.5;
NETWORK
TITLE =
      A     I 34.6;
      AN    I 34.7;
      =     M 26.6;
NETWORK
TITLE =
      A     I 34.7;
      AN    I 34.6;
      =     M 26.7;
NETWORK
TITLE =
      A     I 34.4;
      =     M 21.0;
NETWORK
TITLE =
      A     I 2.2;
      =     M 23.5;
NETWORK
TITLE =
      A     I 32.0;
      FP    M 1000.6;
      =     M 12.1;
NETWORK
TITLE =
      A     M 24.4;
      FP    M 1000.7;
      =     M 25.7;
NETWORK
TITLE =
      A     I 34.0;
      =     M 24.4;
NETWORK
TITLE =
      A     I 35.3;
      =     M 24.5;
NETWORK
TITLE =
      A     M 1.1;
      =     L 2.0;
      A     L 2.0;
      A     DB21.DBX 394.0;
      =     M 25.0;
      A     L 2.0;
      AN    DB21.DBX 394.0;
      =     M 25.1;
NETWORK
TITLE =
      A     I 35.0;
      AN    I 35.1;
      =     M 24.0;
NETWORK
TITLE =
      A     I 35.1;
      AN    I 35.0;
      =     M 24.1;
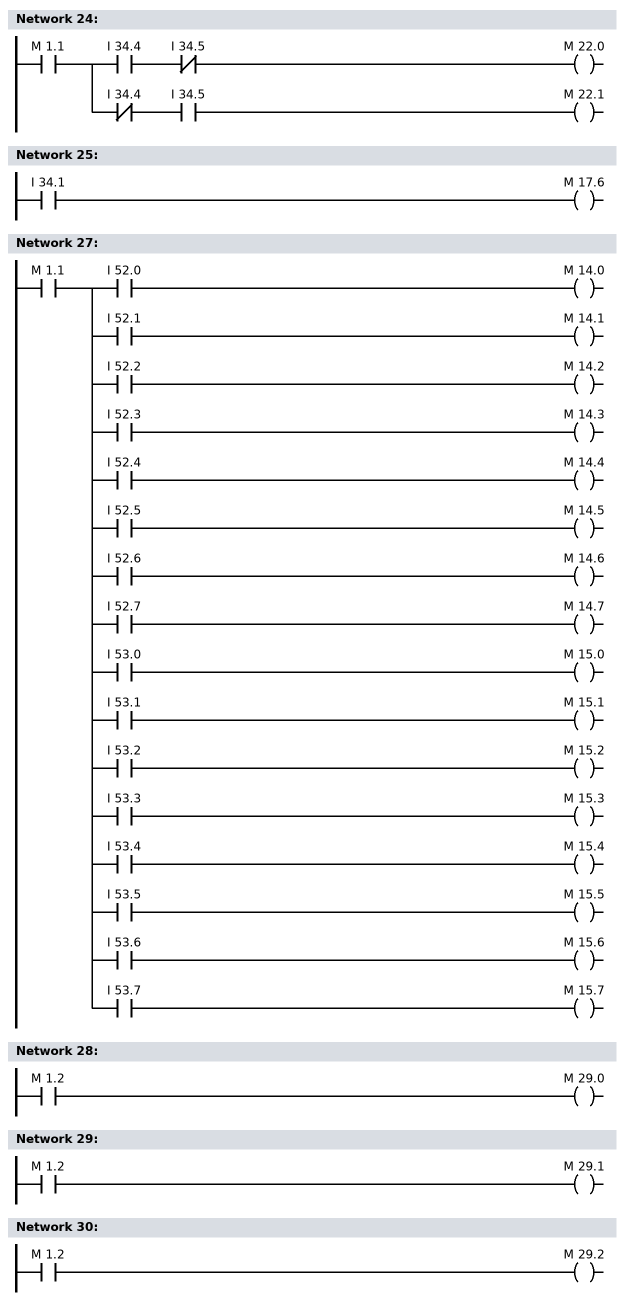
NETWORK
TITLE =
      A     M 1.1;
      =     L 2.0;
      A     L 2.0;
      A     I 34.4;
      AN    I 34.5;
      =     M 22.0;
      A     L 2.0;
      AN    I 34.4;
      A     I 34.5;
      =     M 22.1;
NETWORK
TITLE =
      A     I 34.1;
      =     M 17.6;
NETWORK
TITLE =
NETWORK
TITLE =
      A     M 1.1;
      =     L 2.0;
      A     L 2.0;
      A     I 52.0;
      =     M 14.0;
      A     L 2.0;
      A     I 52.1;
      =     M 14.1;
      A     L 2.0;
      A     I 52.2;
      =     M 14.2;
      A     L 2.0;
      A     I 52.3;
      =     M 14.3;
      A     L 2.0;
      A     I 52.4;
      =     M 14.4;
      A     L 2.0;
      A     I 52.5;
      =     M 14.5;
      A     L 2.0;
      A     I 52.6;
      =     M 14.6;
      A     L 2.0;
      A     I 52.7;
      =     M 14.7;
      A     L 2.0;
      A     I 53.0;
      =     M 15.0;
      A     L 2.0;
      A     I 53.1;
      =     M 15.1;
      A     L 2.0;
      A     I 53.2;
      =     M 15.2;
      A     L 2.0;
      A     I 53.3;
      =     M 15.3;
      A     L 2.0;
      A     I 53.4;
      =     M 15.4;
      A     L 2.0;
      A     I 53.5;
      =     M 15.5;
      A     L 2.0;
      A     I 53.6;
      =     M 15.6;
      A     L 2.0;
      A     I 53.7;
      =     M 15.7;
NETWORK
TITLE =
      A     M 1.2;
      =     M 29.0;
NETWORK
TITLE =
      A     M 1.2;
      =     M 29.1;
NETWORK
TITLE =
      A     M 1.2;
      =     M 29.2;
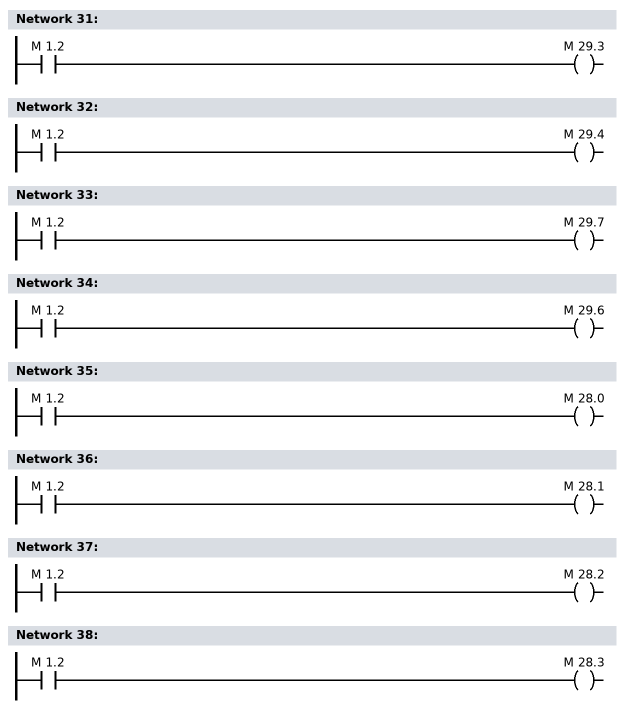
NETWORK
TITLE =
      A     M 1.2;
      =     M 29.3;
NETWORK
TITLE =
      A     M 1.2;
      =     M 29.4;
NETWORK
TITLE =
      A     M 1.2;
      =     M 29.7;
NETWORK
TITLE =
      A     M 1.2;
      =     M 29.6;
NETWORK
TITLE =
      A     M 1.2;
      =     M 28.0;
NETWORK
TITLE =
      A     M 1.2;
      =     M 28.1;
NETWORK
TITLE =
      A     M 1.2;
      =     M 28.2;
NETWORK
TITLE =
      A     M 1.2;
      =     M 28.3;
END_FUNCTION

FUNCTION FC 12 : VOID
VERSION : 0.1
BEGIN
// (block stored without names or comments; labels and parameter names are numbered)
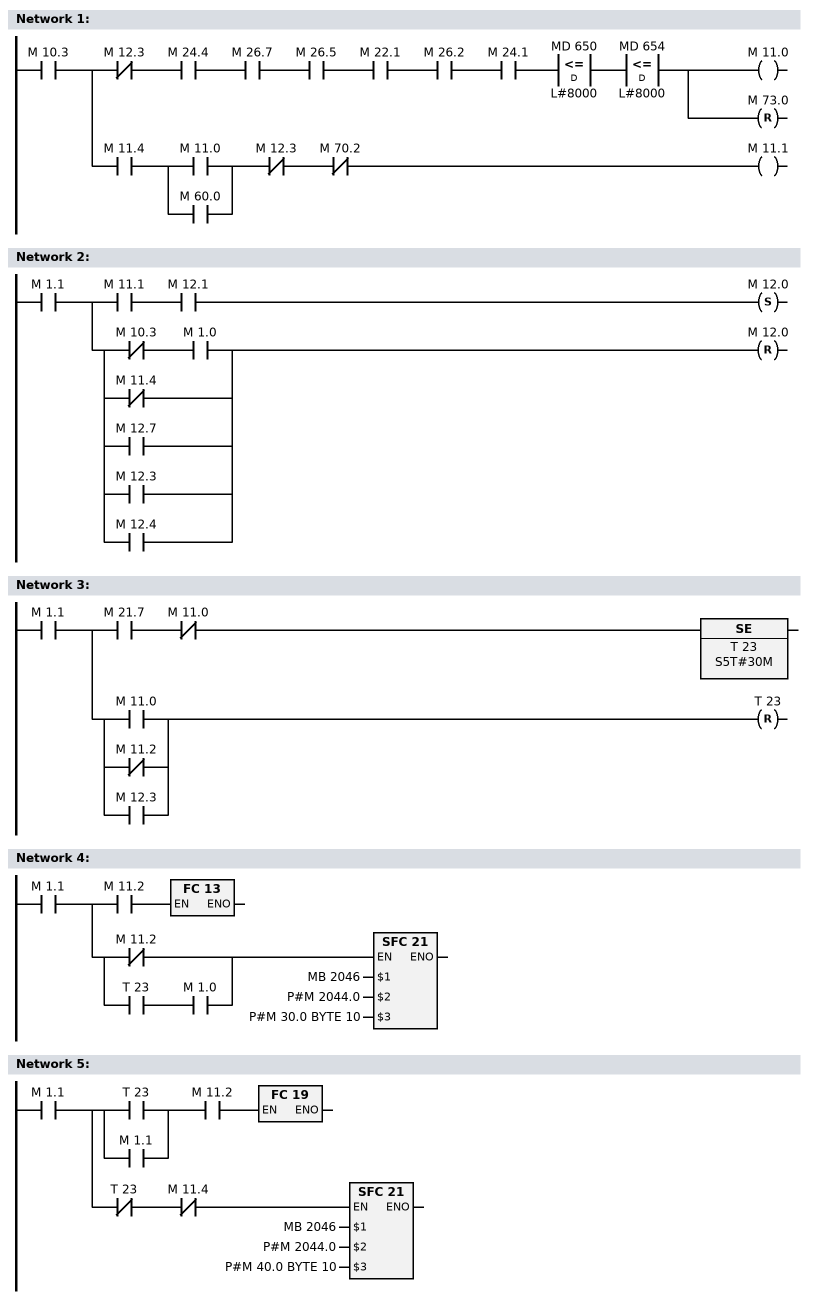
NETWORK
TITLE =
      A     M 10.3;
      =     L 0.0;
      A     L 0.0;
      AN    M 12.3;
      A     M 24.4;
      A     M 26.7;
      A     M 26.5;
      A     M 22.1;
      A     M 26.2;
      A     M 24.1;
      A(;
      L     MD 650;
      L     L#8000;
      <=D;
      );
      A(;
      L     MD 654;
      L     L#8000;
      <=D;
      );
      =     M 11.0;
      R     M 73.0;
      A     L 0.0;
      A     M 11.4;
      A(;
      O     M 11.0;
      O     M 60.0;
      );
      AN    M 12.3;
      AN    M 70.2;
      =     M 11.1;
NETWORK
TITLE =
      A     M 1.1;
      =     L 0.0;
      A     L 0.0;
      A     M 11.1;
      A     M 12.1;
      S     M 12.0;
      A     L 0.0;
      A(;
      AN    M 10.3;
      A     M 1.0;
      ON    M 11.4;
      O     M 12.7;
      O     M 12.3;
      O     M 12.4;
      );
      R     M 12.0;
NETWORK
TITLE =
      A     M 1.1;
      =     L 0.0;
      A     L 0.0;
      A     M 21.7;
      AN    M 11.0;
      L     S5T#30M;
      SE    T 23;
      A     L 0.0;
      A(;
      O     M 11.0;
      ON    M 11.2;
      O     M 12.3;
      );
      R     T 23;
NETWORK
TITLE =
      A     M 1.1;
      =     L 0.0;
      A     L 0.0;
      A     M 11.2;
      JNB   M001;
      CALL  FC 13;
M001: NOP   0;
      A     L 0.0;
      A(;
      ON    M 11.2;
      O;
      A     T 23;
      A     M 1.0;
      );
      JNB   M002;
      CALL  SFC 21 (
           $1                       := MB 2046,
           $2                       := P#M 2044.0,
           $3                       := P#M 30.0 BYTE 10);
M002: NOP   0;
NETWORK
TITLE =
      A     M 1.1;
      =     L 0.0;
      A     L 0.0;
      A(;
      O     T 23;
      O     M 1.1;
      );
      A     M 11.2;
      JNB   M003;
      CALL  FC 19;
M003: NOP   0;
      A     L 0.0;
      AN    T 23;
      AN    M 11.4;
      JNB   M004;
      CALL  SFC 21 (
           $1                       := MB 2046,
           $2                       := P#M 2044.0,
           $3                       := P#M 40.0 BYTE 10);
M004: NOP   0;
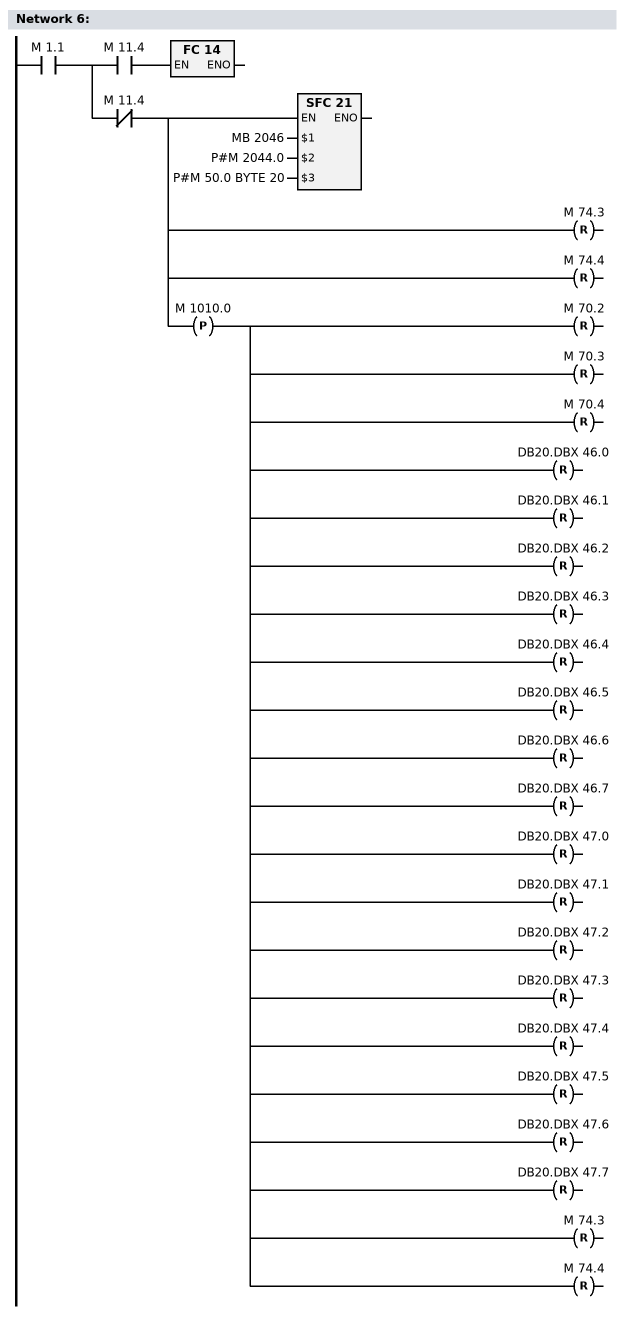
NETWORK
TITLE =
      A     M 1.1;
      =     L 0.0;
      A     L 0.0;
      A     M 11.4;
      JNB   M005;
      CALL  FC 14;
M005: NOP   0;
      A     L 0.0;
      AN    M 11.4;
      =     L 0.1;
      A     L 0.1;
      JNB   M006;
      CALL  SFC 21 (
           $1                       := MB 2046,
           $2                       := P#M 2044.0,
           $3                       := P#M 50.0 BYTE 20);
M006: NOP   0;
      A     L 0.1;
      BLD   102;
      R     M 74.3;
      A     L 0.1;
      BLD   102;
      R     M 74.4;
      A     L 0.1;
      FP    M 1010.0;
      R     M 70.2;
      R     M 70.3;
      R     M 70.4;
      R     DB20.DBX 46.0;
      R     DB20.DBX 46.1;
      R     DB20.DBX 46.2;
      R     DB20.DBX 46.3;
      R     DB20.DBX 46.4;
      R     DB20.DBX 46.5;
      R     DB20.DBX 46.6;
      R     DB20.DBX 46.7;
      R     DB20.DBX 47.0;
      R     DB20.DBX 47.1;
      R     DB20.DBX 47.2;
      R     DB20.DBX 47.3;
      R     DB20.DBX 47.4;
      R     DB20.DBX 47.5;
      R     DB20.DBX 47.6;
      R     DB20.DBX 47.7;
      R     M 74.3;
      R     M 74.4;
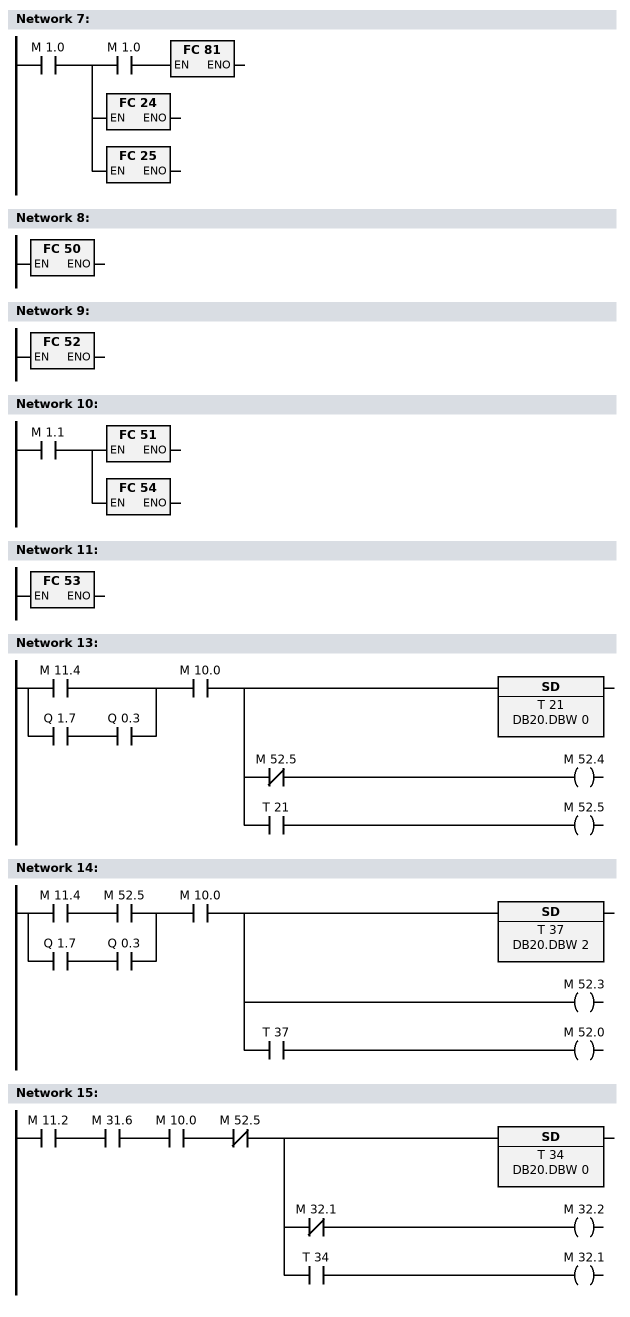
NETWORK
TITLE =
      A     M 1.0;
      =     L 0.0;
      A     L 0.0;
      A     M 1.0;
      JNB   M007;
      CALL  FC 81;
M007: NOP   0;
      A     L 0.0;
      JNB   M008;
      CALL  FC 24;
M008: NOP   0;
      A     L 0.0;
      JNB   M009;
      CALL  FC 25;
M009: NOP   0;
NETWORK
TITLE =
      CALL  FC 50;
      NOP   0;
NETWORK
TITLE =
      CALL  FC 52;
      NOP   0;
NETWORK
TITLE =
      A     M 1.1;
      =     L 0.0;
      A     L 0.0;
      JNB   M010;
      CALL  FC 51;
M010: NOP   0;
      A     L 0.0;
      JNB   M011;
      CALL  FC 54;
M011: NOP   0;
NETWORK
TITLE =
      CALL  FC 53;
      NOP   0;
NETWORK
TITLE =
NETWORK
TITLE =
      A(;
      O     M 11.4;
      O;
      A     Q 1.7;
      A     Q 0.3;
      );
      A     M 10.0;
      =     L 0.0;
      A     L 0.0;
      BLD   102;
      L     DB20.DBW 0;
      SD    T 21;
      A     L 0.0;
      AN    M 52.5;
      =     M 52.4;
      A     L 0.0;
      A     T 21;
      =     M 52.5;
NETWORK
TITLE =
      A(;
      A     M 11.4;
      A     M 52.5;
      O;
      A     Q 1.7;
      A     Q 0.3;
      );
      A     M 10.0;
      =     L 0.0;
      A     L 0.0;
      BLD   102;
      L     DB20.DBW 2;
      SD    T 37;
      A     L 0.0;
      BLD   102;
      =     M 52.3;
      A     L 0.0;
      A     T 37;
      =     M 52.0;
NETWORK
TITLE =
      A     M 11.2;
      A     M 31.6;
      A     M 10.0;
      AN    M 52.5;
      =     L 0.0;
      A     L 0.0;
      BLD   102;
      L     DB20.DBW 0;
      SD    T 34;
      A     L 0.0;
      AN    M 32.1;
      =     M 32.2;
      A     L 0.0;
      A     T 34;
      =     M 32.1;
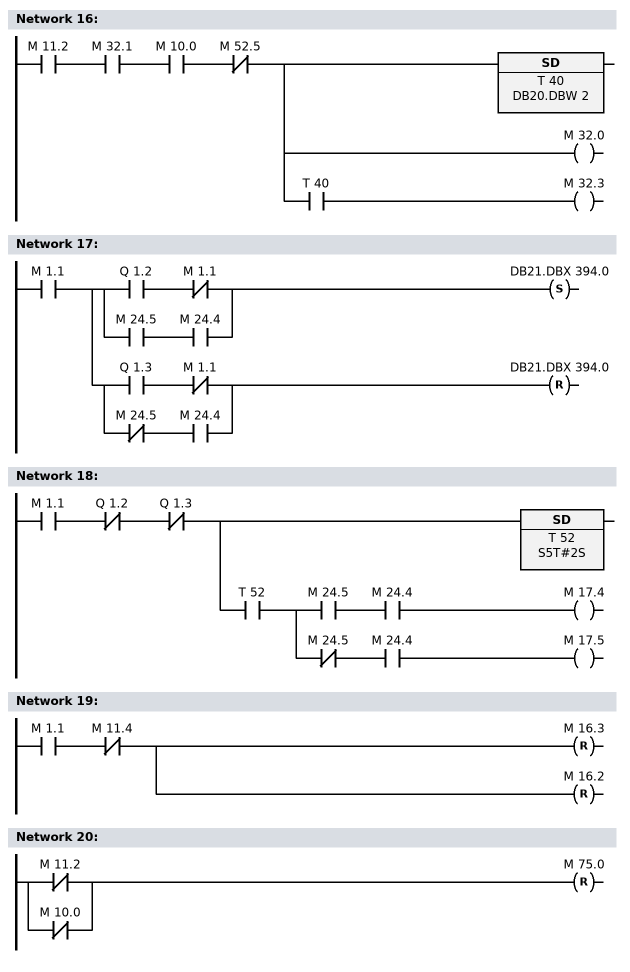
NETWORK
TITLE =
      A     M 11.2;
      A     M 32.1;
      A     M 10.0;
      AN    M 52.5;
      =     L 0.0;
      A     L 0.0;
      BLD   102;
      L     DB20.DBW 2;
      SD    T 40;
      A     L 0.0;
      BLD   102;
      =     M 32.0;
      A     L 0.0;
      A     T 40;
      =     M 32.3;
NETWORK
TITLE =
      A     M 1.1;
      =     L 0.0;
      A     L 0.0;
      A(;
      A     Q 1.2;
      AN    M 1.1;
      O;
      A     M 24.5;
      A     M 24.4;
      );
      S     DB21.DBX 394.0;
      A     L 0.0;
      A(;
      A     Q 1.3;
      AN    M 1.1;
      O;
      AN    M 24.5;
      A     M 24.4;
      );
      R     DB21.DBX 394.0;
NETWORK
TITLE =
      A     M 1.1;
      AN    Q 1.2;
      AN    Q 1.3;
      =     L 0.0;
      A     L 0.0;
      BLD   102;
      L     S5T#2S;
      SD    T 52;
      A     L 0.0;
      A     T 52;
      =     L 0.1;
      A     L 0.1;
      A     M 24.5;
      A     M 24.4;
      =     M 17.4;
      A     L 0.1;
      AN    M 24.5;
      A     M 24.4;
      =     M 17.5;
NETWORK
TITLE =
      A     M 1.1;
      AN    M 11.4;
      R     M 16.3;
      R     M 16.2;
NETWORK
TITLE =
      ON    M 11.2;
      ON    M 10.0;
      R     M 75.0;
END_FUNCTION

FUNCTION FC 13 : VOID
VERSION : 0.1
BEGIN
// (block stored without names or comments; labels and parameter names are numbered)
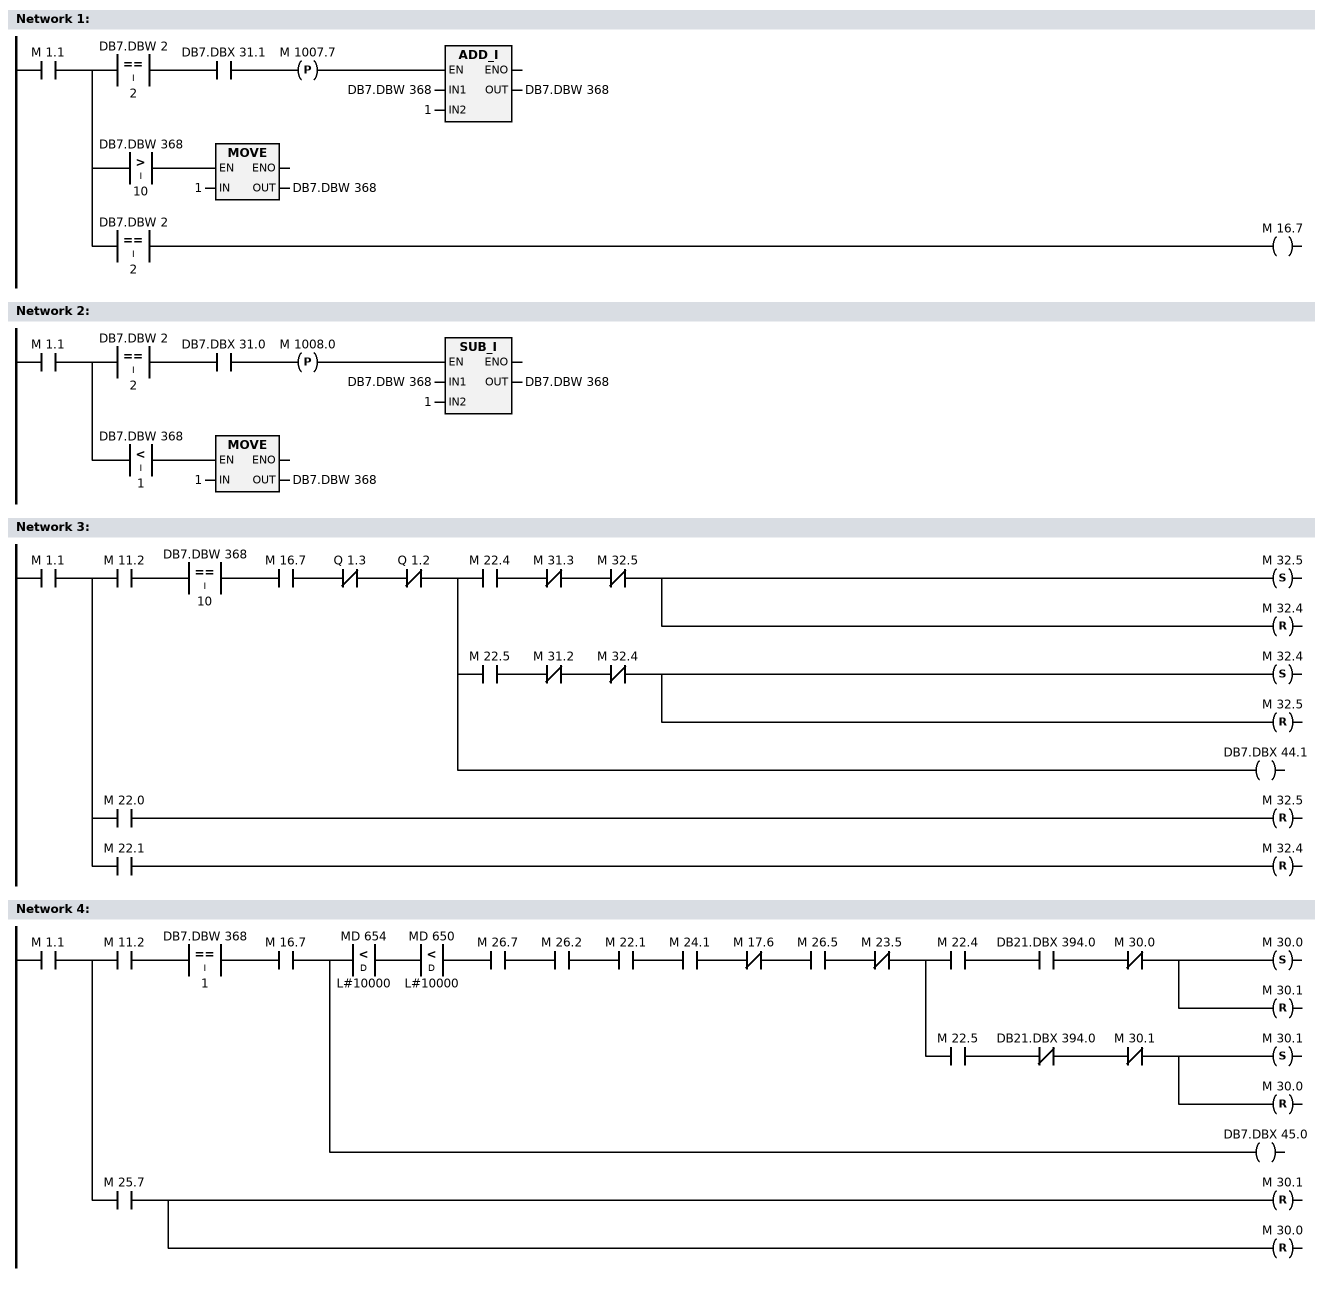
NETWORK
TITLE =
      A     M 1.1;
      =     L 0.0;
      A     L 0.0;
      A(;
      L     DB7.DBW 2;
      L     2;
      ==I;
      );
      A     DB7.DBX 31.1;
      FP    M 1007.7;
      JNB   M001;
      L     DB7.DBW 368;
      L     1;
      +I;
      T     DB7.DBW 368;
M001: NOP   0;
      A     L 0.0;
      A(;
      L     DB7.DBW 368;
      L     10;
      >I;
      );
      JNB   M002;
      L     1;
      T     DB7.DBW 368;
M002: NOP   0;
      A     L 0.0;
      A(;
      L     DB7.DBW 2;
      L     2;
      ==I;
      );
      =     M 16.7;
NETWORK
TITLE =
      A     M 1.1;
      =     L 0.0;
      A     L 0.0;
      A(;
      L     DB7.DBW 2;
      L     2;
      ==I;
      );
      A     DB7.DBX 31.0;
      FP    M 1008.0;
      JNB   M003;
      L     DB7.DBW 368;
      L     1;
      -I;
      T     DB7.DBW 368;
M003: NOP   0;
      A     L 0.0;
      A(;
      L     DB7.DBW 368;
      L     1;
      <I;
      );
      JNB   M004;
      L     1;
      T     DB7.DBW 368;
M004: NOP   0;
NETWORK
TITLE =
      A     M 1.1;
      =     L 0.0;
      A     L 0.0;
      A     M 11.2;
      A(;
      L     DB7.DBW 368;
      L     10;
      ==I;
      );
      A     M 16.7;
      AN    Q 1.3;
      AN    Q 1.2;
      =     L 0.1;
      A     L 0.1;
      A     M 22.4;
      AN    M 31.3;
      AN    M 32.5;
      S     M 32.5;
      R     M 32.4;
      A     L 0.1;
      A     M 22.5;
      AN    M 31.2;
      AN    M 32.4;
      S     M 32.4;
      R     M 32.5;
      A     L 0.1;
      BLD   102;
      =     DB7.DBX 44.1;
      A     L 0.0;
      A     M 22.0;
      R     M 32.5;
      A     L 0.0;
      A     M 22.1;
      R     M 32.4;
NETWORK
TITLE =
      A     M 1.1;
      =     L 0.0;
      A     L 0.0;
      A     M 11.2;
      A(;
      L     DB7.DBW 368;
      L     1;
      ==I;
      );
      A     M 16.7;
      =     L 0.1;
      A     L 0.1;
      A(;
      L     MD 654;
      L     L#10000;
      <D;
      );
      A(;
      L     MD 650;
      L     L#10000;
      <D;
      );
      A     M 26.7;
      A     M 26.2;
      A     M 22.1;
      A     M 24.1;
      AN    M 17.6;
      A     M 26.5;
      AN    M 23.5;
      =     L 0.2;
      A     L 0.2;
      A     M 22.4;
      A     DB21.DBX 394.0;
      AN    M 30.0;
      S     M 30.0;
      R     M 30.1;
      A     L 0.2;
      A     M 22.5;
      AN    DB21.DBX 394.0;
      AN    M 30.1;
      S     M 30.1;
      R     M 30.0;
      A     L 0.1;
      BLD   102;
      =     DB7.DBX 45.0;
      A     L 0.0;
      A     M 25.7;
      R     M 30.1;
      R     M 30.0;
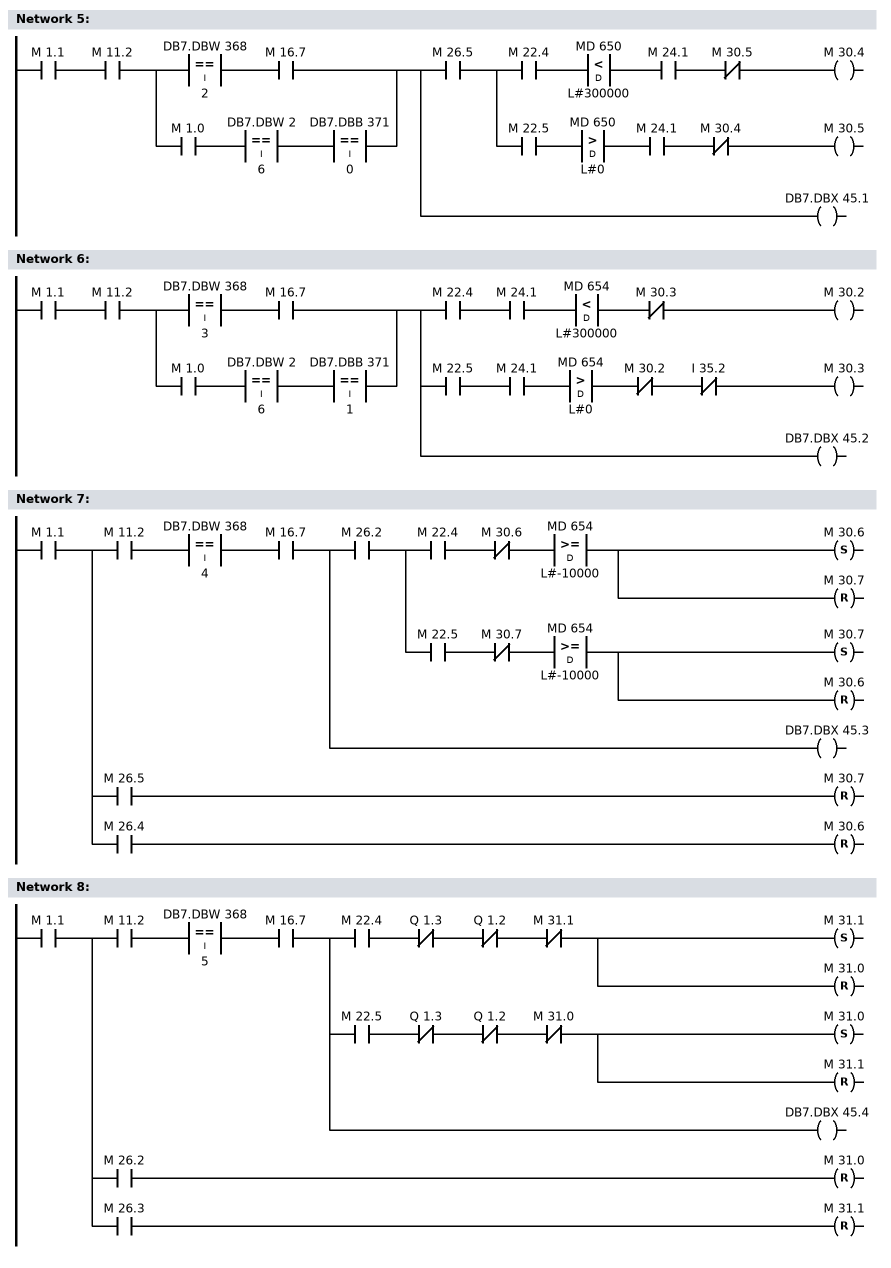
NETWORK
TITLE =
      A     M 1.1;
      A     M 11.2;
      A(;
      A(;
      L     DB7.DBW 368;
      L     2;
      ==I;
      );
      A     M 16.7;
      O;
      A     M 1.0;
      A(;
      L     DB7.DBW 2;
      L     6;
      ==I;
      );
      A(;
      L     DB7.DBB 371;
      L     0;
      ==I;
      );
      );
      =     L 0.0;
      A     L 0.0;
      A     M 26.5;
      =     L 0.1;
      A     L 0.1;
      A     M 22.4;
      A(;
      L     MD 650;
      L     L#300000;
      <D;
      );
      A     M 24.1;
      AN    M 30.5;
      =     M 30.4;
      A     L 0.1;
      A     M 22.5;
      A(;
      L     MD 650;
      L     L#0;
      >D;
      );
      A     M 24.1;
      AN    M 30.4;
      =     M 30.5;
      A     L 0.0;
      BLD   102;
      =     DB7.DBX 45.1;
NETWORK
TITLE =
      A     M 1.1;
      A     M 11.2;
      A(;
      A(;
      L     DB7.DBW 368;
      L     3;
      ==I;
      );
      A     M 16.7;
      O;
      A     M 1.0;
      A(;
      L     DB7.DBW 2;
      L     6;
      ==I;
      );
      A(;
      L     DB7.DBB 371;
      L     1;
      ==I;
      );
      );
      =     L 0.0;
      A     L 0.0;
      A     M 22.4;
      A     M 24.1;
      A(;
      L     MD 654;
      L     L#300000;
      <D;
      );
      AN    M 30.3;
      =     M 30.2;
      A     L 0.0;
      A     M 22.5;
      A     M 24.1;
      A(;
      L     MD 654;
      L     L#0;
      >D;
      );
      AN    M 30.2;
      AN    I 35.2;
      =     M 30.3;
      A     L 0.0;
      BLD   102;
      =     DB7.DBX 45.2;
NETWORK
TITLE =
      A     M 1.1;
      =     L 0.0;
      A     L 0.0;
      A     M 11.2;
      A(;
      L     DB7.DBW 368;
      L     4;
      ==I;
      );
      A     M 16.7;
      =     L 0.1;
      A     L 0.1;
      A     M 26.2;
      =     L 0.2;
      A     L 0.2;
      A     M 22.4;
      AN    M 30.6;
      A(;
      L     MD 654;
      L     L#-10000;
      >=D;
      );
      S     M 30.6;
      R     M 30.7;
      A     L 0.2;
      A     M 22.5;
      AN    M 30.7;
      A(;
      L     MD 654;
      L     L#-10000;
      >=D;
      );
      S     M 30.7;
      R     M 30.6;
      A     L 0.1;
      BLD   102;
      =     DB7.DBX 45.3;
      A     L 0.0;
      A     M 26.5;
      R     M 30.7;
      A     L 0.0;
      A     M 26.4;
      R     M 30.6;
NETWORK
TITLE =
      A     M 1.1;
      =     L 0.0;
      A     L 0.0;
      A     M 11.2;
      A(;
      L     DB7.DBW 368;
      L     5;
      ==I;
      );
      A     M 16.7;
      =     L 0.1;
      A     L 0.1;
      A     M 22.4;
      AN    Q 1.3;
      AN    Q 1.2;
      AN    M 31.1;
      S     M 31.1;
      R     M 31.0;
      A     L 0.1;
      A     M 22.5;
      AN    Q 1.3;
      AN    Q 1.2;
      AN    M 31.0;
      S     M 31.0;
      R     M 31.1;
      A     L 0.1;
      BLD   102;
      =     DB7.DBX 45.4;
      A     L 0.0;
      A     M 26.2;
      R     M 31.0;
      A     L 0.0;
      A     M 26.3;
      R     M 31.1;
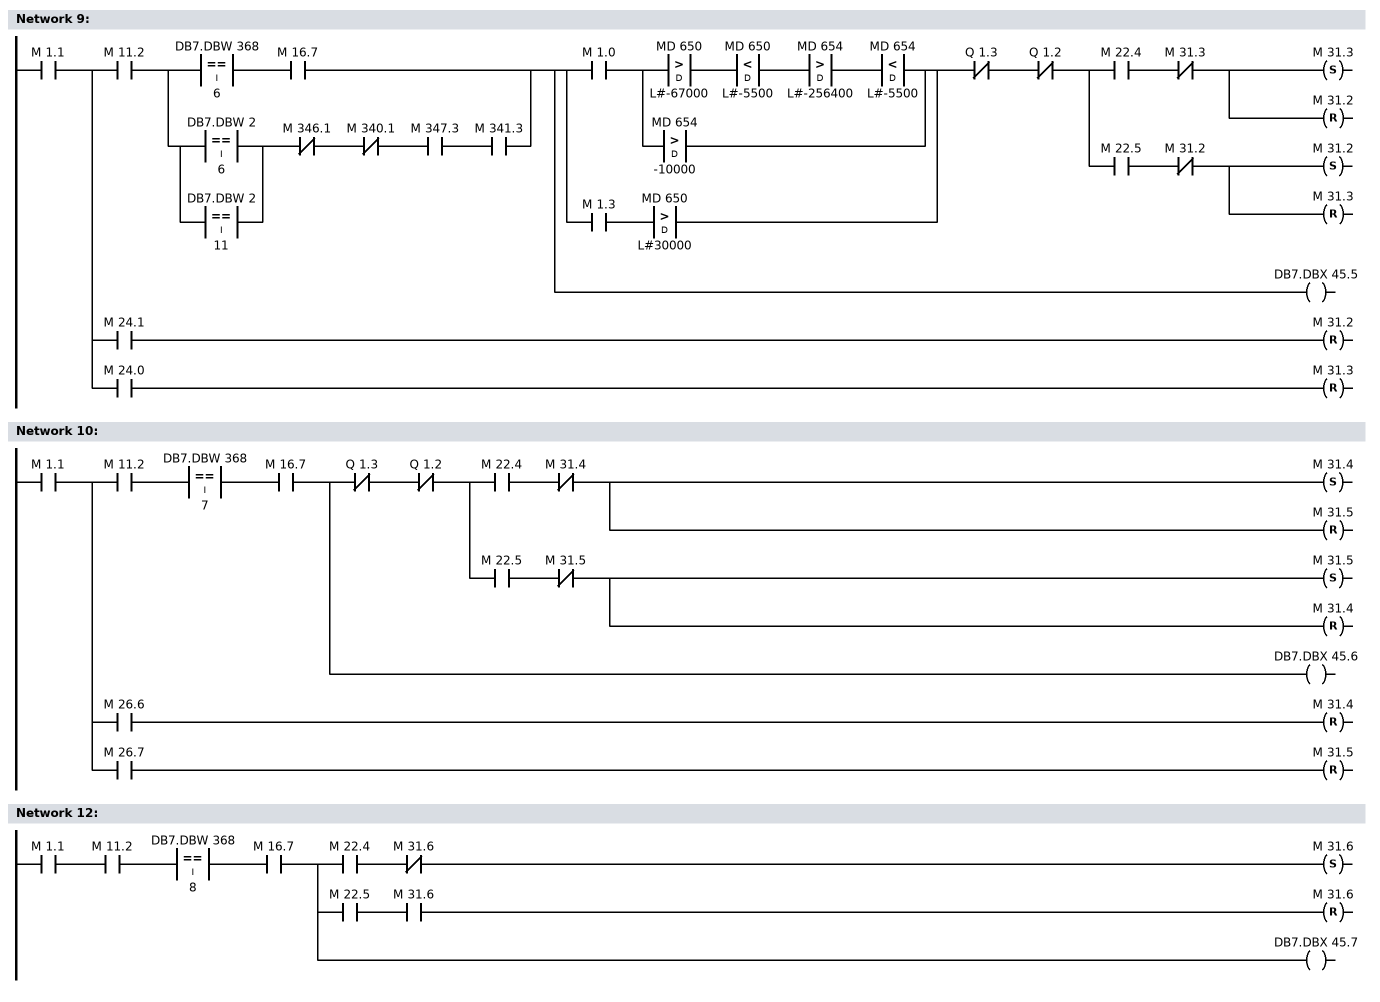
NETWORK
TITLE =
      A     M 1.1;
      =     L 0.0;
      A     L 0.0;
      A     M 11.2;
      A(;
      A(;
      L     DB7.DBW 368;
      L     6;
      ==I;
      );
      A     M 16.7;
      O;
      A(;
      O(;
      L     DB7.DBW 2;
      L     6;
      ==I;
      );
      O(;
      L     DB7.DBW 2;
      L     11;
      ==I;
      );
      );
      AN    M 346.1;
      AN    M 340.1;
      A     M 347.3;
      A     M 341.3;
      );
      =     L 0.1;
      A     L 0.1;
      A(;
      A     M 1.0;
      A(;
      A(;
      L     MD 650;
      L     L#-67000;
      >D;
      );
      A(;
      L     MD 650;
      L     L#-5500;
      <D;
      );
      A(;
      L     MD 654;
      L     L#-256400;
      >D;
      );
      A(;
      L     MD 654;
      L     L#-5500;
      <D;
      );
      O(;
      L     MD 654;
      L     -10000;
      >D;
      );
      );
      O;
      A     M 1.3;
      A(;
      L     MD 650;
      L     L#30000;
      >D;
      );
      );
      AN    Q 1.3;
      AN    Q 1.2;
      =     L 0.2;
      A     L 0.2;
      A     M 22.4;
      AN    M 31.3;
      S     M 31.3;
      R     M 31.2;
      A     L 0.2;
      A     M 22.5;
      AN    M 31.2;
      S     M 31.2;
      R     M 31.3;
      A     L 0.1;
      BLD   102;
      =     DB7.DBX 45.5;
      A     L 0.0;
      A     M 24.1;
      R     M 31.2;
      A     L 0.0;
      A     M 24.0;
      R     M 31.3;
NETWORK
TITLE =
      A     M 1.1;
      =     L 0.0;
      A     L 0.0;
      A     M 11.2;
      A(;
      L     DB7.DBW 368;
      L     7;
      ==I;
      );
      A     M 16.7;
      =     L 0.1;
      A     L 0.1;
      AN    Q 1.3;
      AN    Q 1.2;
      =     L 0.2;
      A     L 0.2;
      A     M 22.4;
      AN    M 31.4;
      S     M 31.4;
      R     M 31.5;
      A     L 0.2;
      A     M 22.5;
      AN    M 31.5;
      S     M 31.5;
      R     M 31.4;
      A     L 0.1;
      BLD   102;
      =     DB7.DBX 45.6;
      A     L 0.0;
      A     M 26.6;
      R     M 31.4;
      A     L 0.0;
      A     M 26.7;
      R     M 31.5;
NETWORK
TITLE =
NETWORK
TITLE =
      A     M 1.1;
      A     M 11.2;
      A(;
      L     DB7.DBW 368;
      L     8;
      ==I;
      );
      A     M 16.7;
      =     L 0.0;
      A     L 0.0;
      A     M 22.4;
      AN    M 31.6;
      S     M 31.6;
      A     L 0.0;
      A     M 22.5;
      A     M 31.6;
      R     M 31.6;
      A     L 0.0;
      BLD   102;
      =     DB7.DBX 45.7;
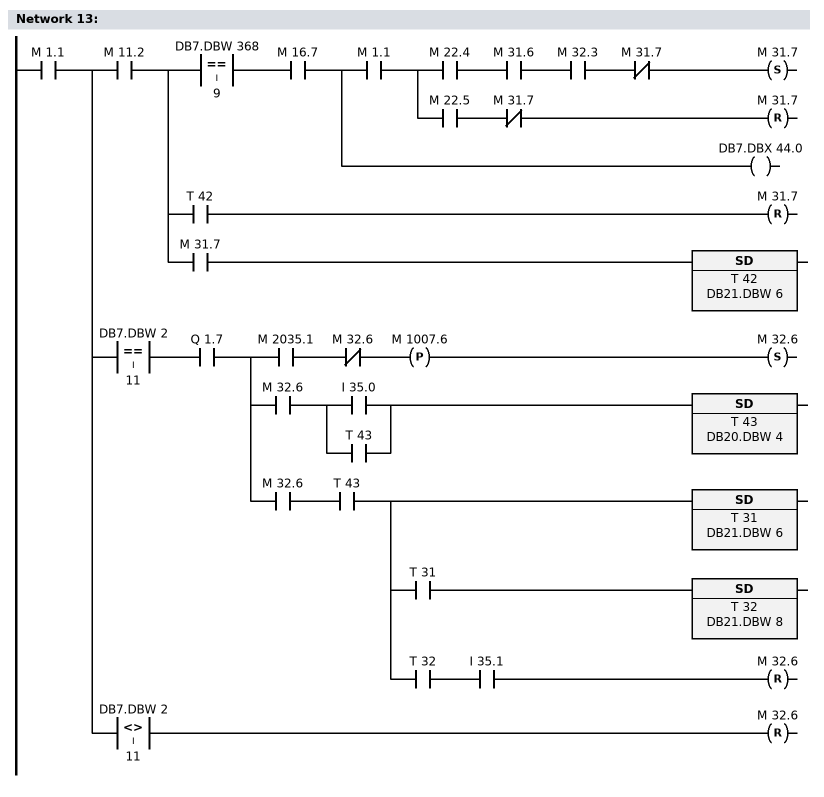
NETWORK
TITLE =
      A     M 1.1;
      =     L 0.0;
      A     L 0.0;
      A     M 11.2;
      =     L 0.1;
      A     L 0.1;
      A(;
      L     DB7.DBW 368;
      L     9;
      ==I;
      );
      A     M 16.7;
      =     L 0.2;
      A     L 0.2;
      A     M 1.1;
      =     L 0.3;
      A     L 0.3;
      A     M 22.4;
      A     M 31.6;
      A     M 32.3;
      AN    M 31.7;
      S     M 31.7;
      A     L 0.3;
      A     M 22.5;
      AN    M 31.7;
      R     M 31.7;
      A     L 0.2;
      BLD   102;
      =     DB7.DBX 44.0;
      A     L 0.1;
      A     T 42;
      R     M 31.7;
      A     L 0.1;
      A     M 31.7;
      L     DB21.DBW 6;
      SD    T 42;
      A     L 0.0;
      A(;
      L     DB7.DBW 2;
      L     11;
      ==I;
      );
      A     Q 1.7;
      =     L 0.1;
      A     L 0.1;
      A     M 2035.1;
      AN    M 32.6;
      FP    M 1007.6;
      S     M 32.6;
      A     L 0.1;
      A     M 32.6;
      A(;
      O     I 35.0;
      O     T 43;
      );
      L     DB20.DBW 4;
      SD    T 43;
      A     L 0.1;
      A     M 32.6;
      A     T 43;
      =     L 0.2;
      A     L 0.2;
      BLD   102;
      L     DB21.DBW 6;
      SD    T 31;
      A     L 0.2;
      A     T 31;
      L     DB21.DBW 8;
      SD    T 32;
      A     L 0.2;
      A     T 32;
      A     I 35.1;
      R     M 32.6;
      A     L 0.0;
      A(;
      L     DB7.DBW 2;
      L     11;
      <>I;
      );
      R     M 32.6;
END_FUNCTION

FUNCTION FC 14 : VOID
VERSION : 0.1
BEGIN
// (block stored without names or comments; labels and parameter names are numbered)
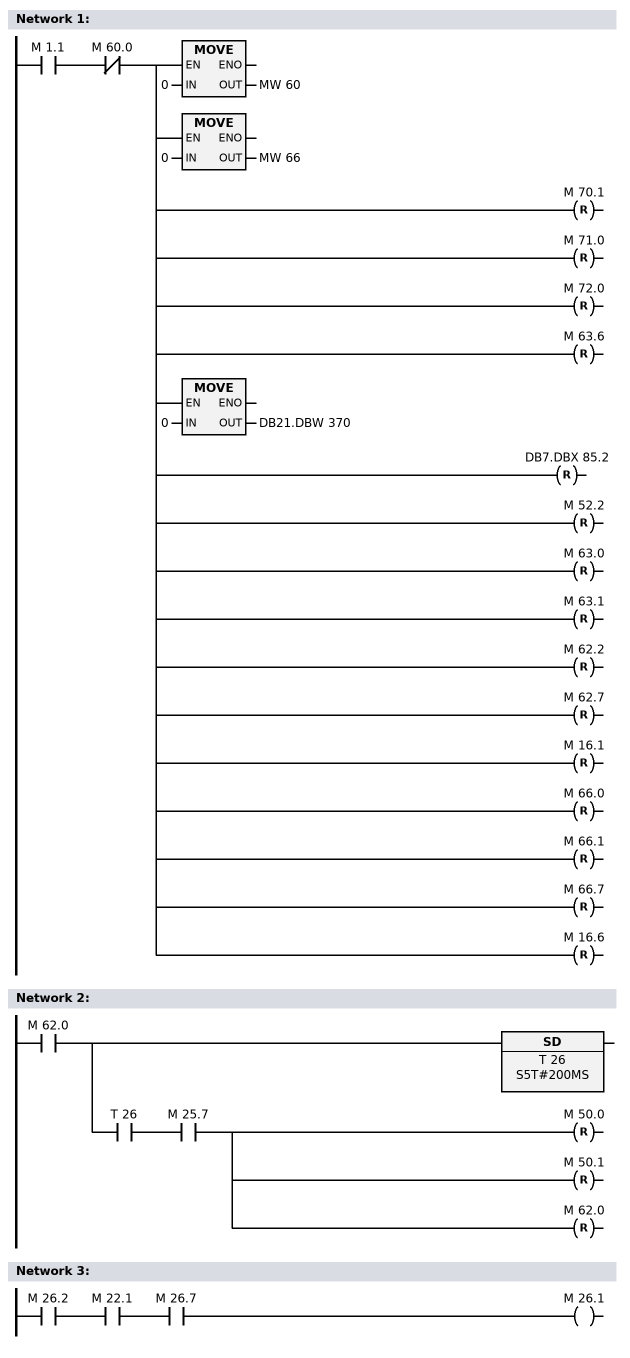
NETWORK
TITLE =
      A     M 1.1;
      AN    M 60.0;
      =     L 24.0;
      A     L 24.0;
      JNB   M001;
      L     0;
      T     MW 60;
M001: NOP   0;
      A     L 24.0;
      JNB   M002;
      L     0;
      T     MW 66;
M002: NOP   0;
      A     L 24.0;
      BLD   102;
      R     M 70.1;
      A     L 24.0;
      BLD   102;
      R     M 71.0;
      A     L 24.0;
      BLD   102;
      R     M 72.0;
      A     L 24.0;
      BLD   102;
      R     M 63.6;
      A     L 24.0;
      JNB   M003;
      L     0;
      T     DB21.DBW 370;
M003: NOP   0;
      A     L 24.0;
      BLD   102;
      R     DB7.DBX 85.2;
      A     L 24.0;
      BLD   102;
      R     M 52.2;
      A     L 24.0;
      BLD   102;
      R     M 63.0;
      A     L 24.0;
      BLD   102;
      R     M 63.1;
      A     L 24.0;
      BLD   102;
      R     M 62.2;
      A     L 24.0;
      BLD   102;
      R     M 62.7;
      A     L 24.0;
      BLD   102;
      R     M 16.1;
      A     L 24.0;
      BLD   102;
      R     M 66.0;
      A     L 24.0;
      BLD   102;
      R     M 66.1;
      A     L 24.0;
      BLD   102;
      R     M 66.7;
      A     L 24.0;
      BLD   102;
      R     M 16.6;
NETWORK
TITLE =
      A     M 62.0;
      =     L 24.0;
      A     L 24.0;
      BLD   102;
      L     S5T#200MS;
      SD    T 26;
      A     L 24.0;
      A     T 26;
      A     M 25.7;
      R     M 50.0;
      R     M 50.1;
      R     M 62.0;
NETWORK
TITLE =
      A     M 26.2;
      A     M 22.1;
      A     M 26.7;
      =     M 26.1;
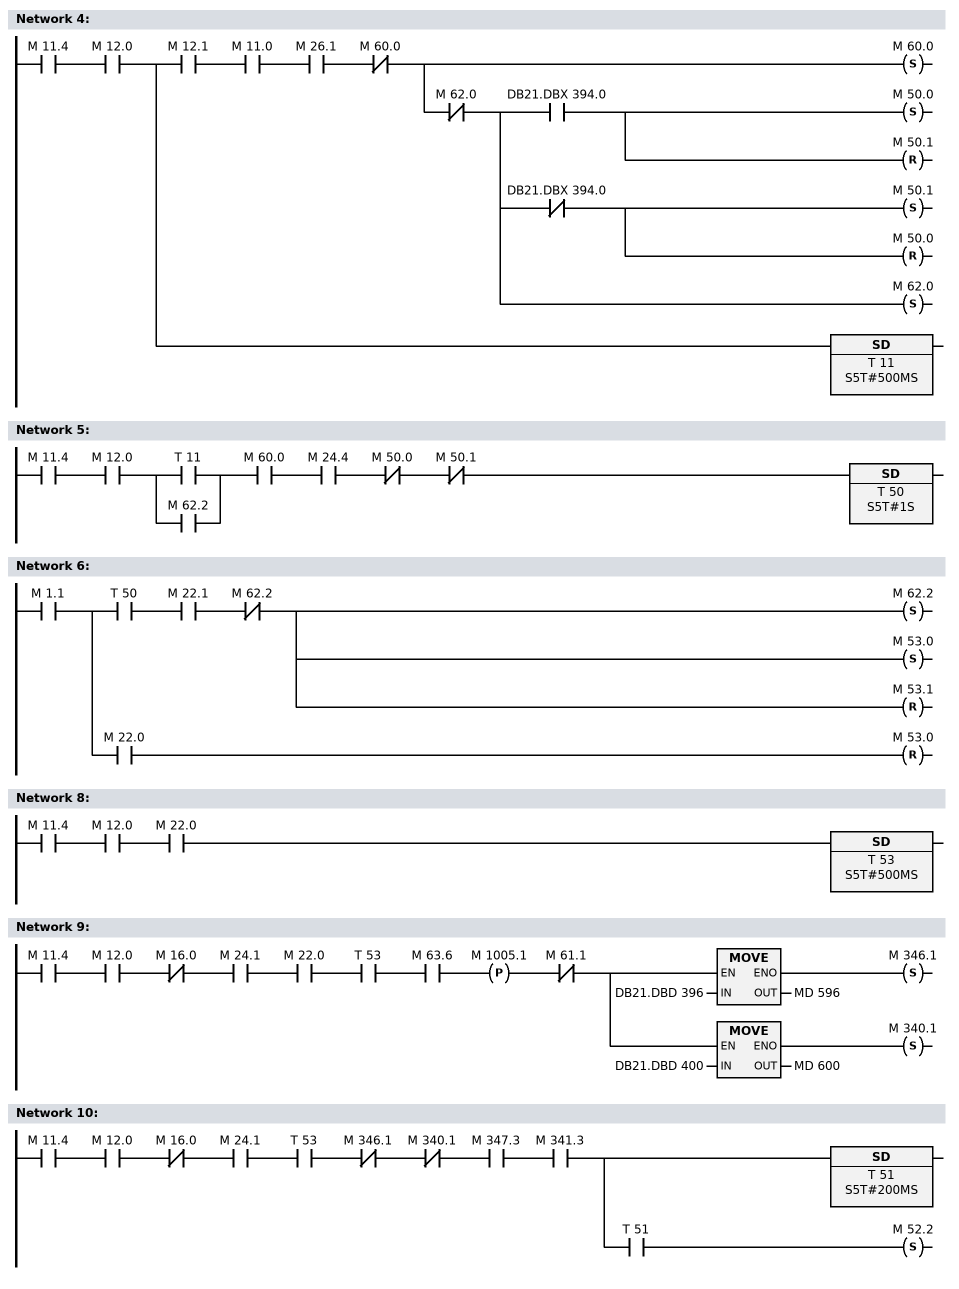
NETWORK
TITLE =
      A     M 11.4;
      A     M 12.0;
      =     L 24.0;
      A     L 24.0;
      A     M 12.1;
      A     M 11.0;
      A     M 26.1;
      AN    M 60.0;
      =     L 24.1;
      A     L 24.1;
      BLD   102;
      S     M 60.0;
      A     L 24.1;
      AN    M 62.0;
      =     L 24.2;
      A     L 24.2;
      A     DB21.DBX 394.0;
      S     M 50.0;
      R     M 50.1;
      A     L 24.2;
      AN    DB21.DBX 394.0;
      S     M 50.1;
      R     M 50.0;
      A     L 24.2;
      BLD   102;
      S     M 62.0;
      A     L 24.0;
      BLD   102;
      L     S5T#500MS;
      SD    T 11;
NETWORK
TITLE =
      A     M 11.4;
      A     M 12.0;
      A(;
      O     T 11;
      O     M 62.2;
      );
      A     M 60.0;
      A     M 24.4;
      AN    M 50.0;
      AN    M 50.1;
      L     S5T#1S;
      SD    T 50;
NETWORK
TITLE =
      A     M 1.1;
      =     L 24.0;
      A     L 24.0;
      A     T 50;
      A     M 22.1;
      AN    M 62.2;
      S     M 62.2;
      S     M 53.0;
      R     M 53.1;
      A     L 24.0;
      A     M 22.0;
      R     M 53.0;
NETWORK
TITLE =
NETWORK
TITLE =
      A     M 11.4;
      A     M 12.0;
      A     M 22.0;
      L     S5T#500MS;
      SD    T 53;
NETWORK
TITLE =
      A     M 11.4;
      A     M 12.0;
      AN    M 16.0;
      A     M 24.1;
      A     M 22.0;
      A     T 53;
      A     M 63.6;
      FP    M 1005.1;
      AN    M 61.1;
      =     L 24.0;
      A     L 24.0;
      JNB   M004;
      L     DB21.DBD 396;
      T     MD 596;
      SET;
      SAVE;
      CLR;
M004: A     BR;
      S     M 346.1;
      A     L 24.0;
      JNB   M005;
      L     DB21.DBD 400;
      T     MD 600;
      SET;
      SAVE;
      CLR;
M005: A     BR;
      S     M 340.1;
NETWORK
TITLE =
      A     M 11.4;
      A     M 12.0;
      AN    M 16.0;
      A     M 24.1;
      A     T 53;
      AN    M 346.1;
      AN    M 340.1;
      A     M 347.3;
      A     M 341.3;
      =     L 24.0;
      A     L 24.0;
      BLD   102;
      L     S5T#200MS;
      SD    T 51;
      A     L 24.0;
      A     T 51;
      S     M 52.2;
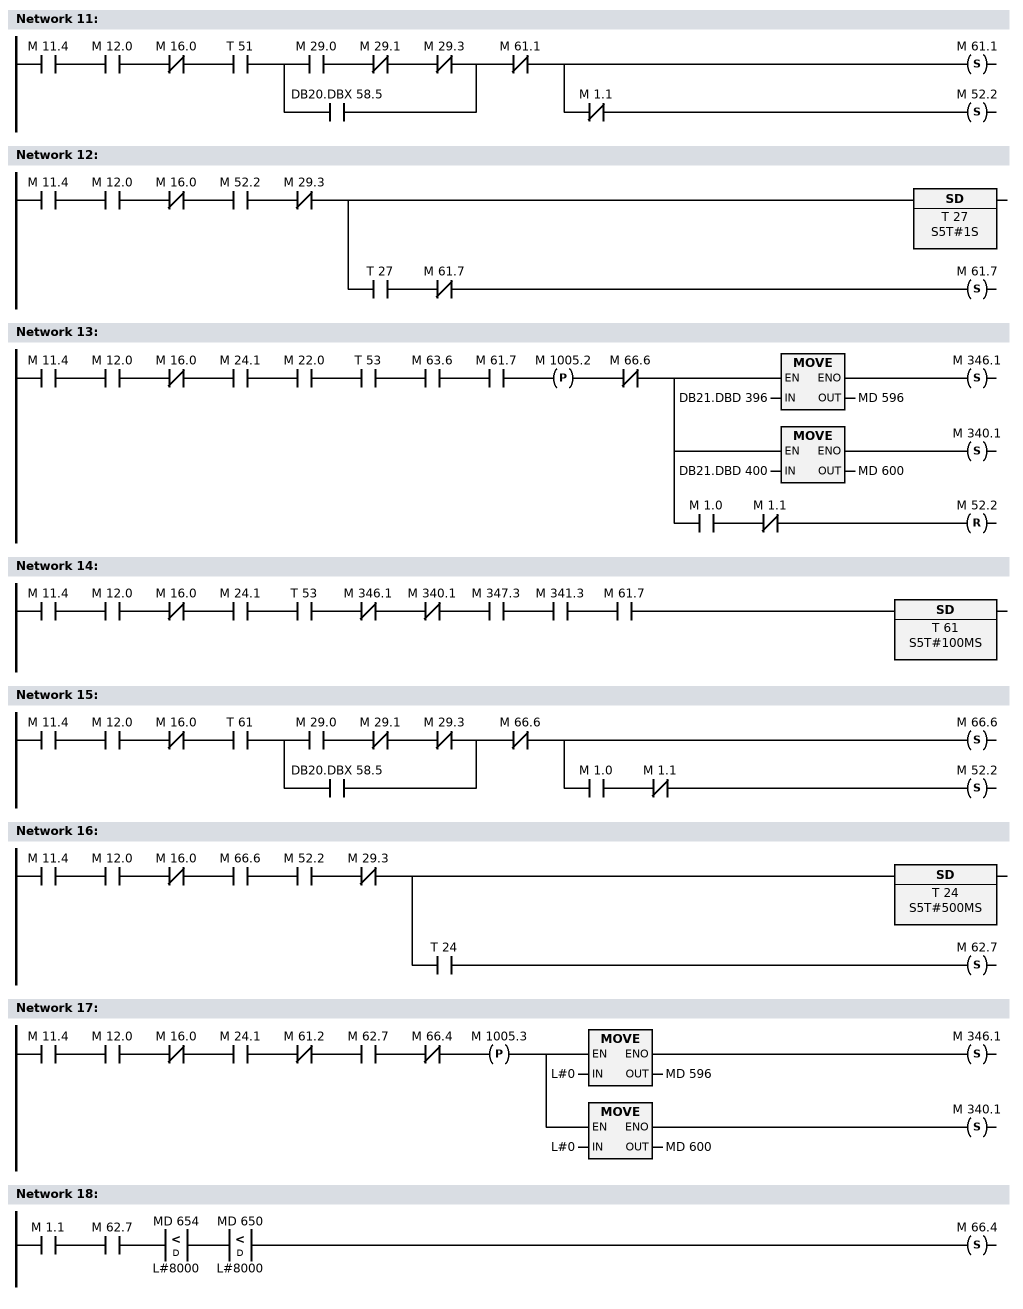
NETWORK
TITLE =
      A     M 11.4;
      A     M 12.0;
      AN    M 16.0;
      A     T 51;
      A(;
      A     M 29.0;
      AN    M 29.1;
      AN    M 29.3;
      O     DB20.DBX 58.5;
      );
      AN    M 61.1;
      =     L 24.0;
      A     L 24.0;
      BLD   102;
      S     M 61.1;
      A     L 24.0;
      AN    M 1.1;
      S     M 52.2;
NETWORK
TITLE =
      A     M 11.4;
      A     M 12.0;
      AN    M 16.0;
      A     M 52.2;
      AN    M 29.3;
      =     L 24.0;
      A     L 24.0;
      BLD   102;
      L     S5T#1S;
      SD    T 27;
      A     L 24.0;
      A     T 27;
      AN    M 61.7;
      S     M 61.7;
NETWORK
TITLE =
      A     M 11.4;
      A     M 12.0;
      AN    M 16.0;
      A     M 24.1;
      A     M 22.0;
      A     T 53;
      A     M 63.6;
      A     M 61.7;
      FP    M 1005.2;
      AN    M 66.6;
      =     L 24.0;
      A     L 24.0;
      JNB   M006;
      L     DB21.DBD 396;
      T     MD 596;
      SET;
      SAVE;
      CLR;
M006: A     BR;
      S     M 346.1;
      A     L 24.0;
      JNB   M007;
      L     DB21.DBD 400;
      T     MD 600;
      SET;
      SAVE;
      CLR;
M007: A     BR;
      S     M 340.1;
      A     L 24.0;
      A     M 1.0;
      AN    M 1.1;
      R     M 52.2;
NETWORK
TITLE =
      A     M 11.4;
      A     M 12.0;
      AN    M 16.0;
      A     M 24.1;
      A     T 53;
      AN    M 346.1;
      AN    M 340.1;
      A     M 347.3;
      A     M 341.3;
      A     M 61.7;
      L     S5T#100MS;
      SD    T 61;
NETWORK
TITLE =
      A     M 11.4;
      A     M 12.0;
      AN    M 16.0;
      A     T 61;
      A(;
      A     M 29.0;
      AN    M 29.1;
      AN    M 29.3;
      O     DB20.DBX 58.5;
      );
      AN    M 66.6;
      =     L 24.0;
      A     L 24.0;
      BLD   102;
      S     M 66.6;
      A     L 24.0;
      A     M 1.0;
      AN    M 1.1;
      S     M 52.2;
NETWORK
TITLE =
      A     M 11.4;
      A     M 12.0;
      AN    M 16.0;
      A     M 66.6;
      A     M 52.2;
      AN    M 29.3;
      =     L 24.0;
      A     L 24.0;
      BLD   102;
      L     S5T#500MS;
      SD    T 24;
      A     L 24.0;
      A     T 24;
      S     M 62.7;
NETWORK
TITLE =
      A     M 11.4;
      A     M 12.0;
      AN    M 16.0;
      A     M 24.1;
      AN    M 61.2;
      A     M 62.7;
      AN    M 66.4;
      FP    M 1005.3;
      =     L 24.0;
      A     L 24.0;
      JNB   M008;
      L     L#0;
      T     MD 596;
      SET;
      SAVE;
      CLR;
M008: A     BR;
      S     M 346.1;
      A     L 24.0;
      JNB   M009;
      L     L#0;
      T     MD 600;
      SET;
      SAVE;
      CLR;
M009: A     BR;
      S     M 340.1;
NETWORK
TITLE =
      A     M 1.1;
      A     M 62.7;
      A(;
      L     MD 654;
      L     L#8000;
      <D;
      );
      A(;
      L     MD 650;
      L     L#8000;
      <D;
      );
      S     M 66.4;
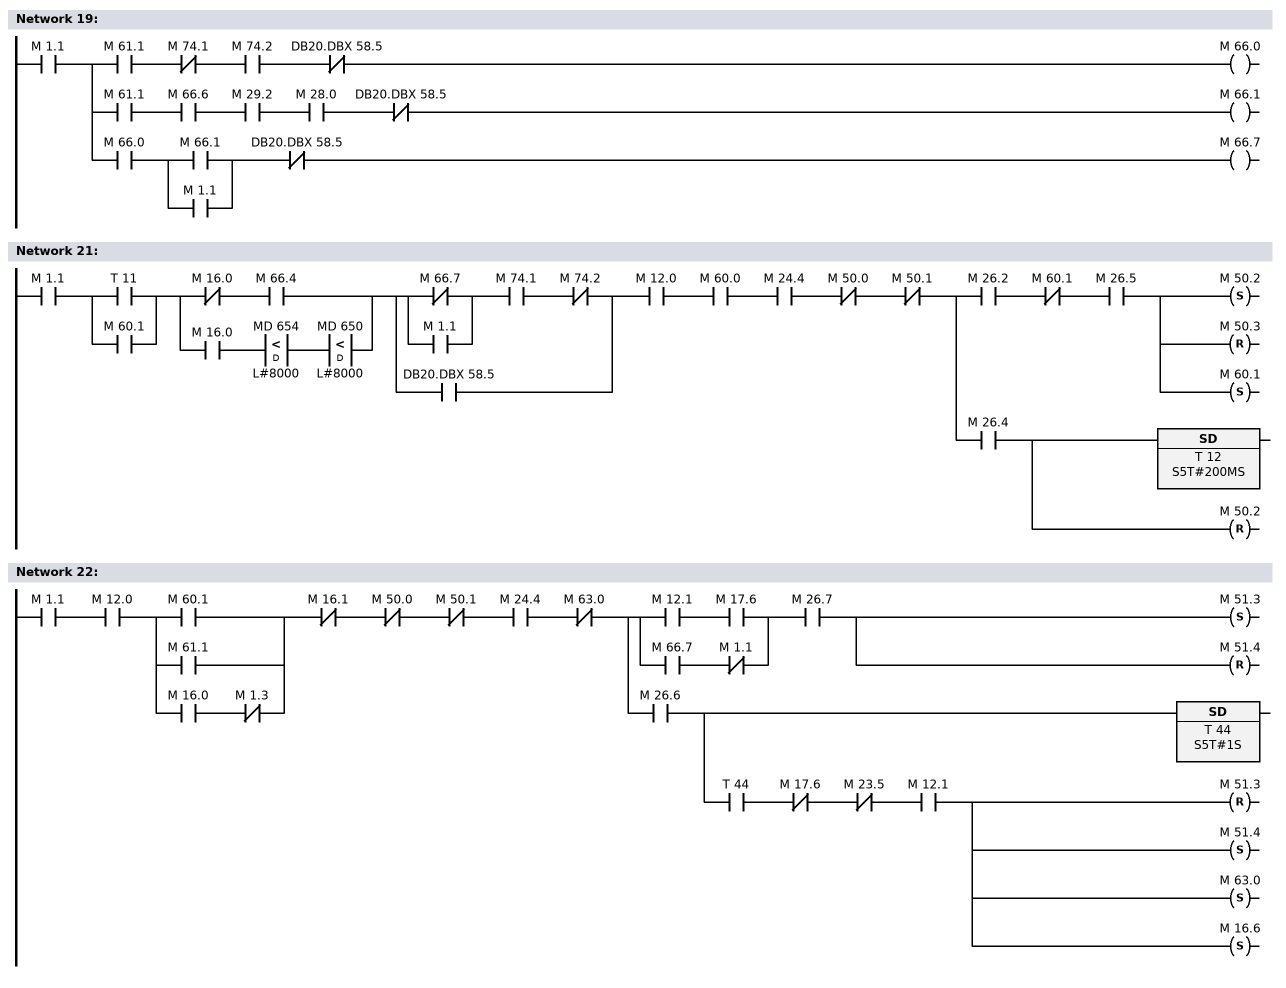
NETWORK
TITLE =
      A     M 1.1;
      =     L 24.0;
      A     L 24.0;
      A     M 61.1;
      AN    M 74.1;
      A     M 74.2;
      AN    DB20.DBX 58.5;
      =     M 66.0;
      A     L 24.0;
      A     M 61.1;
      A     M 66.6;
      A     M 29.2;
      A     M 28.0;
      AN    DB20.DBX 58.5;
      =     M 66.1;
      A     L 24.0;
      A     M 66.0;
      A(;
      O     M 66.1;
      O     M 1.1;
      );
      AN    DB20.DBX 58.5;
      =     M 66.7;
NETWORK
TITLE =
NETWORK
TITLE =
      A     M 1.1;
      A(;
      O     T 11;
      O     M 60.1;
      );
      A(;
      AN    M 16.0;
      A     M 66.4;
      O;
      A     M 16.0;
      A(;
      L     MD 654;
      L     L#8000;
      <D;
      );
      A(;
      L     MD 650;
      L     L#8000;
      <D;
      );
      );
      A(;
      A(;
      ON    M 66.7;
      O     M 1.1;
      );
      A     M 74.1;
      AN    M 74.2;
      O     DB20.DBX 58.5;
      );
      A     M 12.0;
      A     M 60.0;
      A     M 24.4;
      AN    M 50.0;
      AN    M 50.1;
      =     L 24.0;
      A     L 24.0;
      A     M 26.2;
      AN    M 60.1;
      A     M 26.5;
      S     M 50.2;
      R     M 50.3;
      S     M 60.1;
      A     L 24.0;
      A     M 26.4;
      L     S5T#200MS;
      SD    T 12;
      R     M 50.2;
NETWORK
TITLE =
      A     M 1.1;
      A     M 12.0;
      A(;
      O     M 60.1;
      O     M 61.1;
      O;
      A     M 16.0;
      AN    M 1.3;
      );
      AN    M 16.1;
      AN    M 50.0;
      AN    M 50.1;
      A     M 24.4;
      AN    M 63.0;
      =     L 24.0;
      A     L 24.0;
      A(;
      A     M 12.1;
      A     M 17.6;
      O;
      A     M 66.7;
      AN    M 1.1;
      );
      A     M 26.7;
      S     M 51.3;
      R     M 51.4;
      A     L 24.0;
      A     M 26.6;
      =     L 24.1;
      A     L 24.1;
      BLD   102;
      L     S5T#1S;
      SD    T 44;
      A     L 24.1;
      A     T 44;
      AN    M 17.6;
      AN    M 23.5;
      A     M 12.1;
      R     M 51.3;
      S     M 51.4;
      S     M 63.0;
      S     M 16.6;
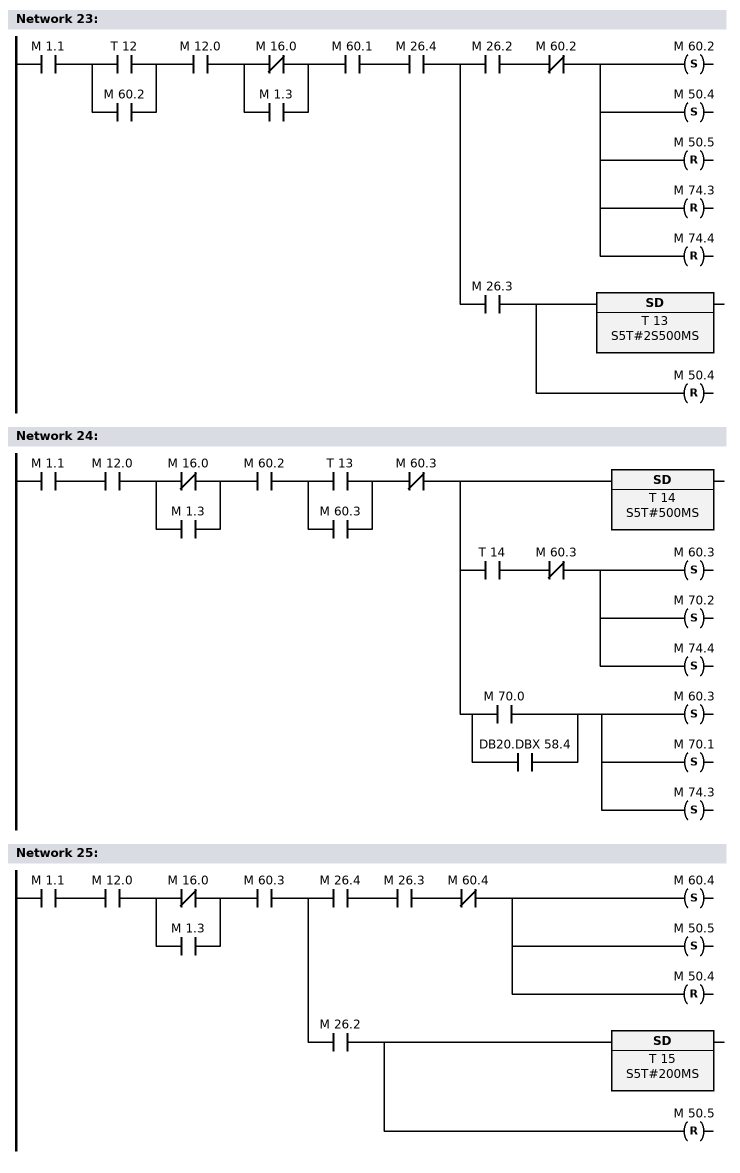
NETWORK
TITLE =
      A     M 1.1;
      A(;
      O     T 12;
      O     M 60.2;
      );
      A     M 12.0;
      A(;
      ON    M 16.0;
      O     M 1.3;
      );
      A     M 60.1;
      A     M 26.4;
      =     L 24.0;
      A     L 24.0;
      A     M 26.2;
      AN    M 60.2;
      S     M 60.2;
      S     M 50.4;
      R     M 50.5;
      R     M 74.3;
      R     M 74.4;
      A     L 24.0;
      A     M 26.3;
      L     S5T#2S500MS;
      SD    T 13;
      R     M 50.4;
NETWORK
TITLE =
      A     M 1.1;
      A     M 12.0;
      A(;
      ON    M 16.0;
      O     M 1.3;
      );
      A     M 60.2;
      A(;
      O     T 13;
      O     M 60.3;
      );
      AN    M 60.3;
      =     L 24.0;
      A     L 24.0;
      BLD   102;
      L     S5T#500MS;
      SD    T 14;
      A     L 24.0;
      A     T 14;
      AN    M 60.3;
      S     M 60.3;
      S     M 70.2;
      S     M 74.4;
      A     L 24.0;
      A(;
      O     M 70.0;
      O     DB20.DBX 58.4;
      );
      S     M 60.3;
      S     M 70.1;
      S     M 74.3;
NETWORK
TITLE =
      A     M 1.1;
      A     M 12.0;
      A(;
      ON    M 16.0;
      O     M 1.3;
      );
      A     M 60.3;
      =     L 24.0;
      A     L 24.0;
      A     M 26.4;
      A     M 26.3;
      AN    M 60.4;
      S     M 60.4;
      S     M 50.5;
      R     M 50.4;
      A     L 24.0;
      A     M 26.2;
      L     S5T#200MS;
      SD    T 15;
      R     M 50.5;
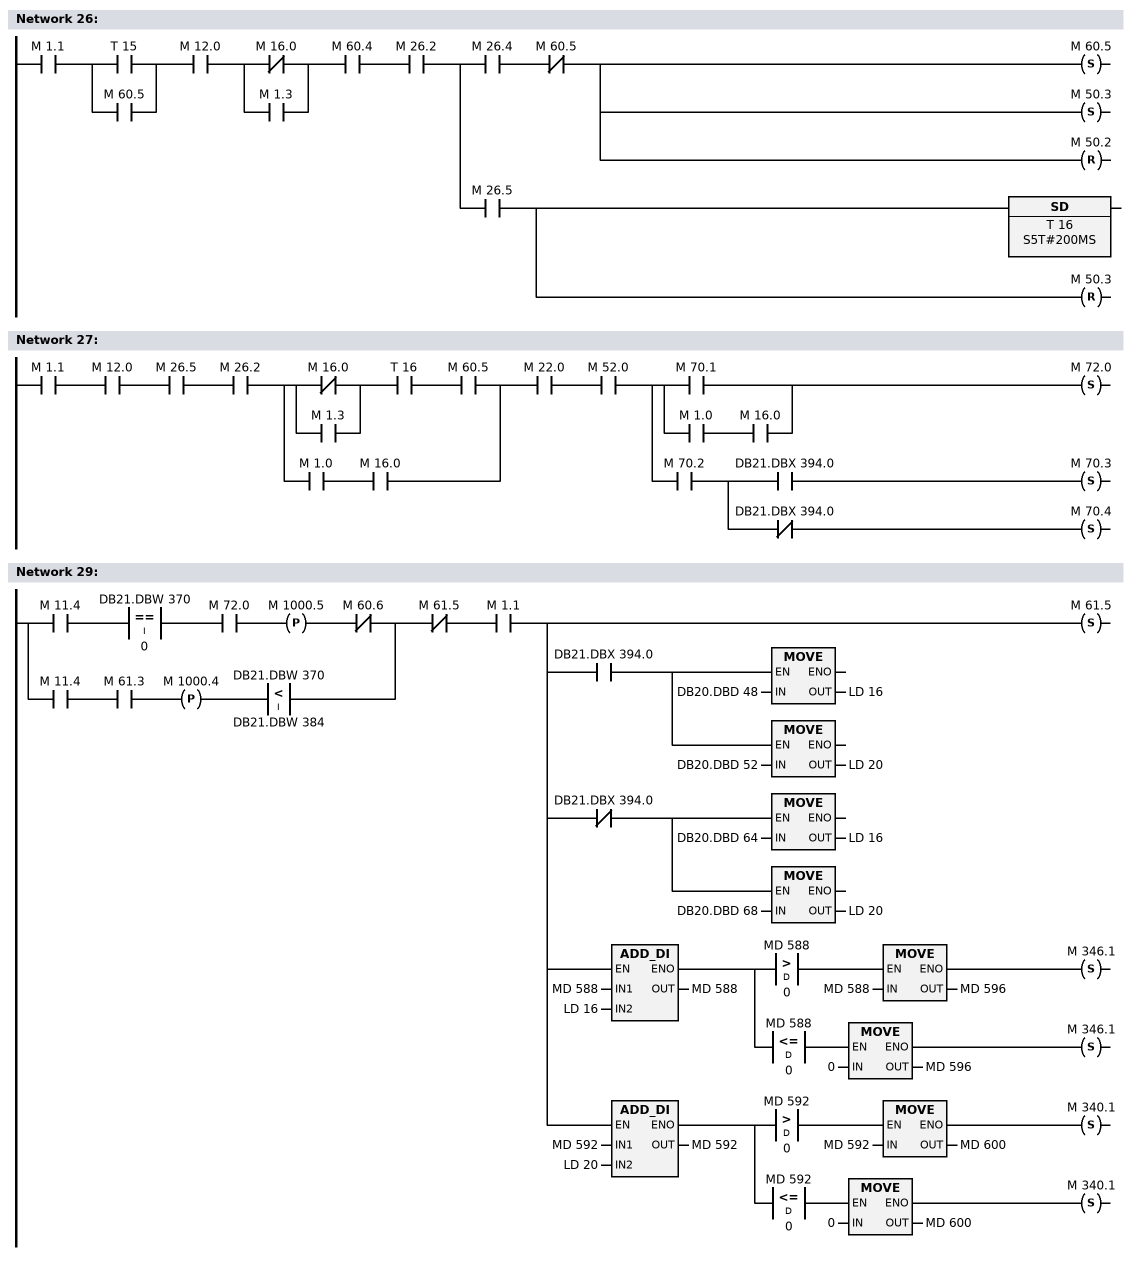
NETWORK
TITLE =
      A     M 1.1;
      A(;
      O     T 15;
      O     M 60.5;
      );
      A     M 12.0;
      A(;
      ON    M 16.0;
      O     M 1.3;
      );
      A     M 60.4;
      A     M 26.2;
      =     L 24.0;
      A     L 24.0;
      A     M 26.4;
      AN    M 60.5;
      S     M 60.5;
      S     M 50.3;
      R     M 50.2;
      A     L 24.0;
      A     M 26.5;
      L     S5T#200MS;
      SD    T 16;
      R     M 50.3;
NETWORK
TITLE =
      A     M 1.1;
      A     M 12.0;
      A     M 26.5;
      A     M 26.2;
      A(;
      A(;
      ON    M 16.0;
      O     M 1.3;
      );
      A     T 16;
      A     M 60.5;
      O;
      A     M 1.0;
      A     M 16.0;
      );
      A     M 22.0;
      A     M 52.0;
      =     L 24.0;
      A     L 24.0;
      A(;
      O     M 70.1;
      O;
      A     M 1.0;
      A     M 16.0;
      );
      S     M 72.0;
      A     L 24.0;
      A     M 70.2;
      =     L 24.1;
      A     L 24.1;
      A     DB21.DBX 394.0;
      S     M 70.3;
      A     L 24.1;
      AN    DB21.DBX 394.0;
      S     M 70.4;
NETWORK
TITLE =
NETWORK
TITLE =
      A(;
      A     M 11.4;
      A(;
      L     DB21.DBW 370;
      L     0;
      ==I;
      );
      A     M 72.0;
      FP    M 1000.5;
      AN    M 60.6;
      O(;
      A     M 11.4;
      A     M 61.3;
      FP    M 1000.4;
      A(;
      L     DB21.DBW 370;
      L     DB21.DBW 384;
      <I;
      );
      );
      );
      AN    M 61.5;
      A     M 1.1;
      =     L 24.0;
      A     L 24.0;
      BLD   102;
      S     M 61.5;
      A     L 24.0;
      A     DB21.DBX 394.0;
      =     L 24.1;
      A     L 24.1;
      JNB   M010;
      L     DB20.DBD 48;
      T     LD 16;
M010: NOP   0;
      A     L 24.1;
      JNB   M011;
      L     DB20.DBD 52;
      T     LD 20;
M011: NOP   0;
      A     L 24.0;
      AN    DB21.DBX 394.0;
      =     L 24.1;
      A     L 24.1;
      JNB   M012;
      L     DB20.DBD 64;
      T     LD 16;
M012: NOP   0;
      A     L 24.1;
      JNB   M013;
      L     DB20.DBD 68;
      T     LD 20;
M013: NOP   0;
      A     L 24.0;
      JNB   M014;
      L     MD 588;
      L     LD 16;
      +D;
      T     MD 588;
      AN    OV;
      SAVE;
      CLR;
M014: A     BR;
      =     L 24.1;
      A     L 24.1;
      A(;
      L     MD 588;
      L     0;
      >D;
      );
      JNB   M015;
      L     MD 588;
      T     MD 596;
      SET;
      SAVE;
      CLR;
M015: A     BR;
      S     M 346.1;
      A     L 24.1;
      A(;
      L     MD 588;
      L     0;
      <=D;
      );
      JNB   M016;
      L     0;
      T     MD 596;
      SET;
      SAVE;
      CLR;
M016: A     BR;
      S     M 346.1;
      A     L 24.0;
      JNB   M017;
      L     MD 592;
      L     LD 20;
      +D;
      T     MD 592;
      AN    OV;
      SAVE;
      CLR;
M017: A     BR;
      =     L 24.1;
      A     L 24.1;
      A(;
      L     MD 592;
      L     0;
      >D;
      );
      JNB   M018;
      L     MD 592;
      T     MD 600;
      SET;
      SAVE;
      CLR;
M018: A     BR;
      S     M 340.1;
      A     L 24.1;
      A(;
      L     MD 592;
      L     0;
      <=D;
      );
      JNB   M019;
      L     0;
      T     MD 600;
      SET;
      SAVE;
      CLR;
M019: A     BR;
      S     M 340.1;
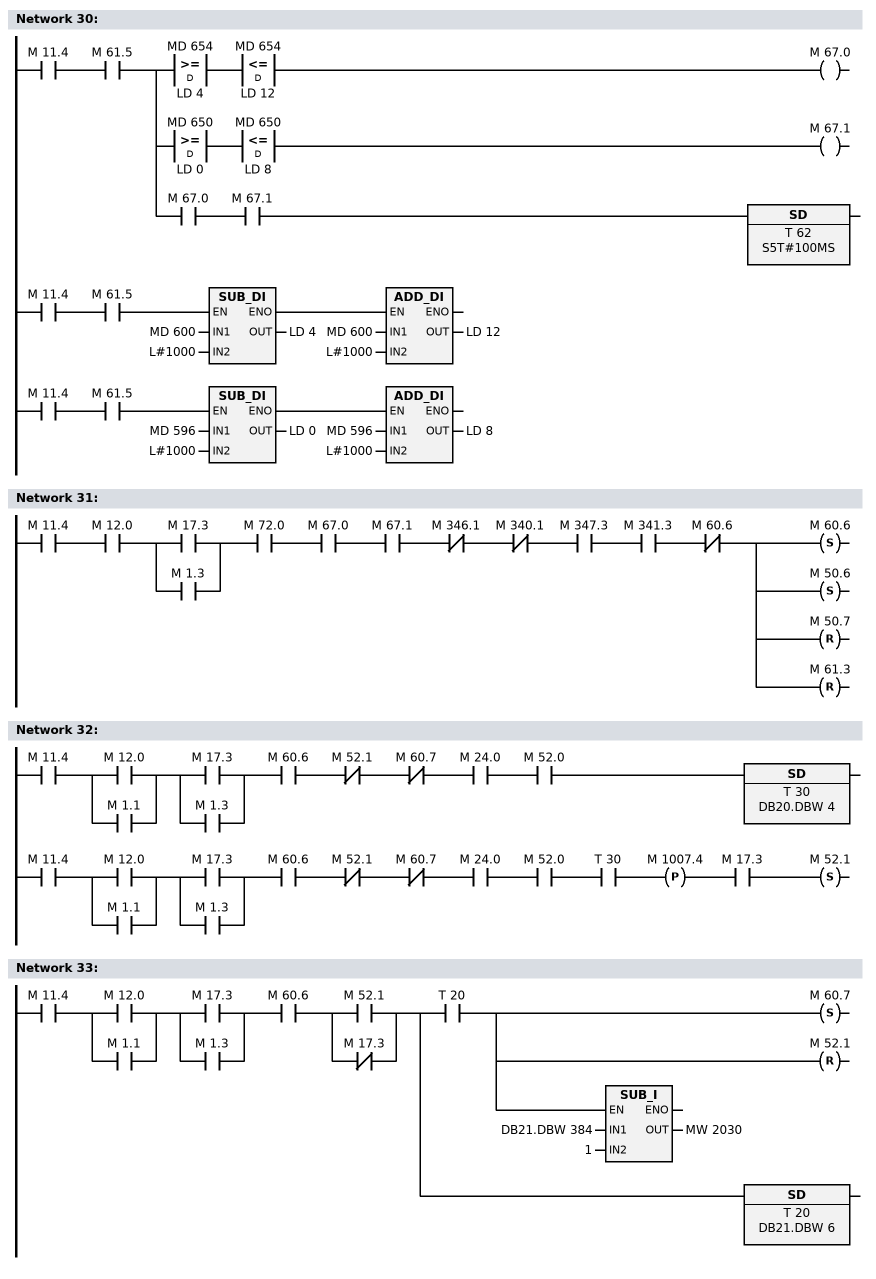
NETWORK
TITLE =
      A     M 11.4;
      A     M 61.5;
      =     L 24.0;
      A(;
      A     L 24.0;
      JNB   M020;
      L     MD 600;
      L     L#1000;
      -D;
      T     LD 4;
      AN    OV;
      SAVE;
      CLR;
M020: A     BR;
      );
      JNB   M021;
      L     MD 600;
      L     L#1000;
      +D;
      T     LD 12;
M021: NOP   0;
      A(;
      A     L 24.0;
      JNB   M022;
      L     MD 596;
      L     L#1000;
      -D;
      T     LD 0;
      AN    OV;
      SAVE;
      CLR;
M022: A     BR;
      );
      JNB   M023;
      L     MD 596;
      L     L#1000;
      +D;
      T     LD 8;
M023: NOP   0;
      A     L 24.0;
      A(;
      L     MD 654;
      L     LD 4;
      >=D;
      );
      A(;
      L     MD 654;
      L     LD 12;
      <=D;
      );
      =     M 67.0;
      A     L 24.0;
      A(;
      L     MD 650;
      L     LD 0;
      >=D;
      );
      A(;
      L     MD 650;
      L     LD 8;
      <=D;
      );
      =     M 67.1;
      A     L 24.0;
      A     M 67.0;
      A     M 67.1;
      L     S5T#100MS;
      SD    T 62;
NETWORK
TITLE =
      A     M 11.4;
      A     M 12.0;
      A(;
      O     M 17.3;
      O     M 1.3;
      );
      A     M 72.0;
      A     M 67.0;
      A     M 67.1;
      AN    M 346.1;
      AN    M 340.1;
      A     M 347.3;
      A     M 341.3;
      AN    M 60.6;
      S     M 60.6;
      S     M 50.6;
      R     M 50.7;
      R     M 61.3;
NETWORK
TITLE =
      A     M 11.4;
      A(;
      O     M 12.0;
      O     M 1.1;
      );
      A(;
      O     M 17.3;
      O     M 1.3;
      );
      A     M 60.6;
      AN    M 52.1;
      AN    M 60.7;
      A     M 24.0;
      A     M 52.0;
      =     L 24.0;
      A     L 24.0;
      BLD   102;
      L     DB20.DBW 4;
      SD    T 30;
      A(;
      A     L 24.0;
      A     T 30;
      FP    M 1007.4;
      );
      A     M 17.3;
      S     M 52.1;
NETWORK
TITLE =
      A     M 11.4;
      A(;
      O     M 12.0;
      O     M 1.1;
      );
      A(;
      O     M 17.3;
      O     M 1.3;
      );
      A     M 60.6;
      A(;
      O     M 52.1;
      ON    M 17.3;
      );
      =     L 24.0;
      A     L 24.0;
      A     T 20;
      =     L 24.1;
      A     L 24.1;
      BLD   102;
      S     M 60.7;
      A     L 24.1;
      BLD   102;
      R     M 52.1;
      A     L 24.1;
      JNB   M024;
      L     DB21.DBW 384;
      L     1;
      -I;
      T     MW 2030;
M024: NOP   0;
      A     L 24.0;
      BLD   102;
      L     DB21.DBW 6;
      SD    T 20;
